CASE eObjectType OF
	E_BACnetObjType.ObjAnalogInput:
		IF ePropID = E_BACnetPropIdentifier.PropPresentValue OR ePropID = E_BACnetPropIdentifier.PropStatusFlags THEN
			F_IsCovProperty:=TRUE;
		END_IF
	E_BACnetObjType.ObjAnalogOutput:
		IF ePropID = E_BACnetPropIdentifier.PropPresentValue OR ePropID = E_BACnetPropIdentifier.PropStatusFlags THEN
			F_IsCovProperty:=TRUE;
		END_IF
	E_BACnetObjType.ObjAnalogValue:
		IF ePropID = E_BACnetPropIdentifier.PropPresentValue OR ePropID = E_BACnetPropIdentifier.PropStatusFlags THEN
			F_IsCovProperty:=TRUE;
		END_IF
	E_BACnetObjType.ObjBinaryInput:
		IF ePropID = E_BACnetPropIdentifier.PropPresentValue OR ePropID = E_BACnetPropIdentifier.PropStatusFlags THEN
			F_IsCovProperty:=TRUE;
		END_IF
	E_BACnetObjType.ObjBinaryOutput:
		IF ePropID = E_BACnetPropIdentifier.PropPresentValue OR ePropID = E_BACnetPropIdentifier.PropStatusFlags THEN
			F_IsCovProperty:=TRUE;
		END_IF
	E_BACnetObjType.ObjBinaryValue:
		IF ePropID = E_BACnetPropIdentifier.PropPresentValue OR ePropID = E_BACnetPropIdentifier.PropStatusFlags THEN
			F_IsCovProperty:=TRUE;
		END_IF
	E_BACnetObjType.ObjMultiStateInput:
		IF ePropID = E_BACnetPropIdentifier.PropPresentValue OR ePropID = E_BACnetPropIdentifier.PropStatusFlags THEN
			F_IsCovProperty:=TRUE;
		END_IF
	E_BACnetObjType.ObjMultiStateOutput:
		IF ePropID = E_BACnetPropIdentifier.PropPresentValue OR ePropID = E_BACnetPropIdentifier.PropStatusFlags THEN
			F_IsCovProperty:=TRUE;
		END_IF
	E_BACnetObjType.ObjMultiStateValue:
		IF ePropID = E_BACnetPropIdentifier.PropPresentValue OR ePropID = E_BACnetPropIdentifier.PropStatusFlags THEN
			F_IsCovProperty:=TRUE;
		END_IF
	E_BACnetObjType.ObjLargeAnalogValue:
		IF ePropID = E_BACnetPropIdentifier.PropPresentValue OR ePropID = E_BACnetPropIdentifier.PropStatusFlags THEN
			F_IsCovProperty:=TRUE;
		END_IF
	E_BACnetObjType.ObjPositiveIntegerValue:
		IF ePropID = E_BACnetPropIdentifier.PropPresentValue OR ePropID = E_BACnetPropIdentifier.PropStatusFlags THEN
			F_IsCovProperty:=TRUE;
		END_IF
	E_BACnetObjType.ObjIntegerValue:
		IF ePropID = E_BACnetPropIdentifier.PropPresentValue OR ePropID = E_BACnetPropIdentifier.PropStatusFlags THEN
			F_IsCovProperty:=TRUE;
		END_IF
	E_BACnetObjType.ObjOctetStringValue:
		IF ePropID = E_BACnetPropIdentifier.PropPresentValue OR ePropID = E_BACnetPropIdentifier.PropStatusFlags THEN
			F_IsCovProperty:=TRUE;
		END_IF
	E_BACnetObjType.ObjCharacterStringValue:
		IF ePropID = E_BACnetPropIdentifier.PropPresentValue OR ePropID = E_BACnetPropIdentifier.PropStatusFlags THEN
			F_IsCovProperty:=TRUE;
		END_IF
	E_BACnetObjType.ObjTimePatternValue:
		IF ePropID = E_BACnetPropIdentifier.PropPresentValue OR ePropID = E_BACnetPropIdentifier.PropStatusFlags THEN
			F_IsCovProperty:=TRUE;
		END_IF
	E_BACnetObjType.ObjTimeValue:
		IF ePropID = E_BACnetPropIdentifier.PropPresentValue OR ePropID = E_BACnetPropIdentifier.PropStatusFlags THEN
			F_IsCovProperty:=TRUE;
		END_IF
	E_BACnetObjType.ObjDatePatternValue:
		IF ePropID = E_BACnetPropIdentifier.PropPresentValue OR ePropID = E_BACnetPropIdentifier.PropStatusFlags THEN
			F_IsCovProperty:=TRUE;
		END_IF
	E_BACnetObjType.ObjDateValue:
		IF ePropID = E_BACnetPropIdentifier.PropPresentValue OR ePropID = E_BACnetPropIdentifier.PropStatusFlags THEN
			F_IsCovProperty:=TRUE;
		END_IF
	E_BACnetObjType.ObjDateTimePatternValue:
		IF ePropID = E_BACnetPropIdentifier.PropPresentValue OR ePropID = E_BACnetPropIdentifier.PropStatusFlags THEN
			F_IsCovProperty:=TRUE;
		END_IF
	E_BACnetObjType.ObjDateTimeValue:
		IF ePropID = E_BACnetPropIdentifier.PropPresentValue OR ePropID = E_BACnetPropIdentifier.PropStatusFlags THEN
			F_IsCovProperty:=TRUE;
		END_IF
	E_BACnetObjType.ObjLoop:
		IF ePropID = E_BACnetPropIdentifier.PropPresentValue OR ePropID = E_BACnetPropIdentifier.PropStatusFlags OR ePropID = E_BACnetPropIdentifier.PropSetpoint OR ePropID = E_BACnetPropIdentifier.PropControlledVariableValue THEN
			F_IsCovProperty:=TRUE;
		END_IF
	E_BACnetObjType.ObjPulseConverter:
			IF ePropID = E_BACnetPropIdentifier.PropPresentValue OR ePropID = E_BACnetPropIdentifier.PropStatusFlags OR ePropID = E_BACnetPropIdentifier.PropUpdateTime THEN
			F_IsCovProperty:=TRUE;
		END_IF
END_CASE

END_FUNCTION

// POUs/Helper/[internal]/Remote/F_IsCovReadMode
{attribute 'hide'}
FUNCTION F_IsCovReadMode : BOOL
VAR_INPUT
	eReadMode : E_BACnet_CommMode;
END_VAR

IF eReadMode = E_BACnet_CommMode.eCov OR eReadMode = E_BACnet_CommMode.eCovC OR eReadMode = E_BACnet_CommMode.eCovU THEN
	F_IsCovReadMode:=TRUE;
END_IF

END_FUNCTION

// POUs/Helper/[internal]/Remote/F_IsCovReqType
{attribute 'hide'}
FUNCTION F_IsCovReqType : BOOL
VAR_INPUT
	iReq : I_BACnetRM_BaseReq;
END_VAR
VAR
	tmpReqType : E_BACnetRM_RequestType;
END_VAR

tmpReqType := iReq.GetRequestType();

IF tmpReqType = E_BACnetRM_RequestType.eCOV OR tmpReqType = E_BACnetRM_RequestType.eCOV_C OR tmpReqType = E_BACnetRM_RequestType.eCOV_U THEN
	F_IsCovReqType:=TRUE;
END_IF

END_FUNCTION

// POUs/Helper/[internal]/Validation-Functions/F_BACnet_IsAbortReasonValid
{attribute 'hide'}
FUNCTION F_BACnet_IsAbortReasonValid : BOOL
VAR_INPUT
	eReason		: E_BACnet_AbortReason;
END_VAR

F_BACnet_IsAbortReasonValid := (E_BACnet_AbortReason.First <= eReason) AND_THEN (eReason <= E_BACnet_AbortReason.Last);

END_FUNCTION

// POUs/Helper/[internal]/Validation-Functions/F_BACnet_IsErrorClassValid
{attribute 'hide'}
FUNCTION F_BACnet_IsErrorClassValid : BOOL
VAR_INPUT
	eClass		: E_BACnet_ErrorClass;
END_VAR

F_BACnet_IsErrorClassValid := (E_BACnet_ErrorClass.First <= eClass) AND_THEN (eClass <= E_BACnet_ErrorClass.Last);

END_FUNCTION

// POUs/Helper/[internal]/Validation-Functions/F_BACnet_IsErrorCodeValid
{attribute 'hide'}
FUNCTION F_BACnet_IsErrorCodeValid : BOOL
VAR_INPUT
	eCode		: E_BACnet_ErrorCode;
END_VAR

F_BACnet_IsErrorCodeValid := (E_BACnet_ErrorCode.First <= eCode) AND_THEN (eCode <= E_BACnet_ErrorCode.Last);

END_FUNCTION

// POUs/Helper/[internal]/Validation-Functions/F_BACnet_IsErrorTypeValid
{attribute 'hide'}
FUNCTION F_BACnet_IsErrorTypeValid : BOOL
VAR_INPUT
	eType		: E_BACnet_ErrorType;
END_VAR

F_BACnet_IsErrorTypeValid := (E_BACnet_ErrorType.First <= eType) AND_THEN (eType <= E_BACnet_ErrorType.Last);

END_FUNCTION

// POUs/Helper/[internal]/Validation-Functions/F_BACnet_IsPropIdentifierValid
{attribute 'hide'}
FUNCTION F_BACnet_IsPropIdentifierValid : BOOL
VAR_INPUT
	eProperty		: E_BACnetPropIdentifier;
END_VAR

F_BACnet_IsPropIdentifierValid := (eProperty <> E_BACnetPropIdentifier.PropInvalid);

END_FUNCTION

// POUs/Helper/[internal]/Validation-Functions/F_BACnet_IsRejectReasonValid
{attribute 'hide'}
FUNCTION F_BACnet_IsRejectReasonValid : BOOL
VAR_INPUT
	eReason		: E_BACnet_RejectReason;
END_VAR

F_BACnet_IsRejectReasonValid := (E_BACnet_RejectReason.First <= eReason) AND_THEN (eReason <= E_BACnet_RejectReason.Last);

END_FUNCTION

// POUs/Helper/[internal]/F_BACnet_AnalogPV
{attribute 'hide'}
FUNCTION F_BACnet_AnalogPV : REAL
VAR_INPUT
	bEnable	: BOOL; (* TRUE = commit to stack, FALSE = do-nothing *)
	bNull	: BOOL; (* TRUE = clear priority, FALSE = write value from input *)
	fValue	: REAL;
END_VAR
VAR
	pres : POINTER TO DWORD;
END_VAR

IF (bEnable) THEN
	IF (bNull) THEN
		pres := ADR(F_BACnet_AnalogPV);
		pres^ := F_BACnet_RealNull(); 
	ELSE
		F_BACnet_AnalogPV := fValue;
	END_IF
ELSE
	F_BACnet_AnalogPV := F_BACnet_NAN();
END_IF

END_FUNCTION

// POUs/Helper/Real/F_BACnet_RealNull
FUNCTION F_BACnet_RealNull : DWORD
(* function that generates <not-a-number> real state *)

F_BACnet_RealNull:=16#7FFF0000;

END_FUNCTION

// POUs/Helper/Real/F_BACnet_NAN
FUNCTION F_BACnet_NAN : REAL
(* function that generates <not-a-number> real state *)
VAR
	res : POINTER TO DWORD;
END_VAR

res:=ADR(F_BACnet_NAN);
res^:=16#7FFFFFFF;

END_FUNCTION

// POUs/Helper/[internal]/F_BACnet_ChangeBitFieldBit
{attribute 'hide'}
FUNCTION F_BACnet_ChangeBitFieldBit : DWORD
VAR_INPUT
	ptrData		: POINTER TO DWORD;
	bitNbr			: INT;
	Value		: BOOL;
END_VAR
VAR
END_VAR

IF (NOT Value) THEN
	ptrData^ := ptrData^ AND NOT (SHR(DWORD#16#00008000,F_BACnet_BitFieldBit(bitNbr)));
ELSE
	ptrData^ := ptrData^ OR (SHR(DWORD#16#00008000,F_BACnet_BitFieldBit(bitNbr)));
END_IF
F_BACnet_ChangeBitFieldBit := ptrData^;

END_FUNCTION

// POUs/Helper/[internal]/F_BACnet_ElemSize
{attribute 'hide'}
FUNCTION F_BACnet_ElemSize : UDINT
VAR_INPUT
	nSize : UDINT;
END_VAR

F_BACnet_ElemSize := (nSize AND 16#7FFFFFFF);

END_FUNCTION

// POUs/Helper/[internal]/F_BACnet_IsBitFieldBitSetPtr
{attribute 'hide'}
FUNCTION F_BACnet_IsBitFieldBitSetPtr : BOOL
VAR_INPUT
	pData	:	POINTER TO WORD;
	bitNbr	:	INT;
END_VAR
VAR
END_VAR

F_BACnet_IsBitFieldBitSetPtr:= ((pData^) AND (SHR(16#8000,F_BACnet_BitFieldBit(bitNbr)))) > 0;

END_FUNCTION

// POUs/Helper/[internal]/F_BACnet_UnSetBitFieldBit
{attribute 'hide'}
FUNCTION F_BACnet_UnSetBitFieldBit : DWORD
VAR_INPUT
	ptrData		:	POINTER TO DWORD;
	bitNbr			:	INT;
END_VAR
VAR
END_VAR

ptrData^ := ptrData^ AND NOT (SHR(DWORD#16#00008000,F_BACnet_BitFieldBit(bitNbr)));
F_BACnet_UnSetBitFieldBit := ptrData^;

END_FUNCTION

// POUs/Helper/Flags/F_BACnet_EventEnable
FUNCTION F_BACnet_EventEnable : UINT
VAR_INPUT
	stEvtEn       : ST_BA_EventTransitions;
END_VAR
VAR
	nEvtEnToFlt     : UINT;
	nEvtEnToNmal    : UINT;
	nEvtEnToOffnmal : UINT;
	nEvtEnNo        : UINT;
END_VAR

(*=============================================*)
(*EventEnable*)
IF	stEvtEn.bToFault
THEN
	nEvtEnToFlt := 16#4000;
ELSE
	nEvtEnToFlt := 16#0;
END_IF

IF	stEvtEn.bToNormal
THEN
	nEvtEnToNmal := 16#2000;
ELSE
	nEvtEnToNmal := 16#0;
END_IF

IF	stEvtEn.bToOffnormal
THEN
	nEvtEnToOffnmal := 16#8000;
ELSE
	nEvtEnToOffnmal := 16#0;
END_IF

nEvtEnNo := 5;

F_BACnet_EventEnable := nEvtEnNo + nEvtEnToFlt + nEvtEnToNmal + nEvtEnToOffnmal;
(*=============================================*)

END_FUNCTION

// POUs/Helper/Flags/F_BACnet_EventTransitionFlags
FUNCTION F_BACnet_EventTransitionFlags : ST_BA_EventTransitions
VAR_INPUT
	data	: WORD;
END_VAR
VAR
END_VAR

F_BACnet_EventTransitionFlags.bToNormal := F_BACnet_IsBitFieldBitSet(data, E_BACnet_EventTransitionBits.eToNormal);
F_BACnet_EventTransitionFlags.bToOffnormal := F_BACnet_IsBitFieldBitSet(data, E_BACnet_EventTransitionBits.eToOffnormal);
F_BACnet_EventTransitionFlags.bToFault := F_BACnet_IsBitFieldBitSet(data, E_BACnet_EventTransitionBits.eToFault);

END_FUNCTION

// POUs/Helper/Flags/F_BACnet_GetEventTransFlagsData
FUNCTION F_BACnet_GetEventTransFlagsData : WORD
VAR_INPUT
	Flags	: ST_BA_EventTransitions;
END_VAR
VAR
END_VAR

F_BACnet_GetEventTransFlagsData := 16#0005;
IF Flags.bToNormal THEN
	F_BACnet_GetEventTransFlagsData := DWORD_TO_WORD(F_BACnet_SetBitFieldBit(ptrData:=ADR(F_BACnet_GetEventTransFlagsData), bitNbr:=E_BACnet_EventTransitionBits.eToNormal));
END_IF
IF Flags.bToOffnormal THEN
	F_BACnet_GetEventTransFlagsData := DWORD_TO_WORD(F_BACnet_SetBitFieldBit(ptrData:=ADR(F_BACnet_GetEventTransFlagsData), bitNbr:=E_BACnet_EventTransitionBits.eToOffnormal));
END_IF
IF Flags.bToFault THEN
	F_BACnet_GetEventTransFlagsData := DWORD_TO_WORD(F_BACnet_SetBitFieldBit(ptrData:=ADR(F_BACnet_GetEventTransFlagsData), bitNbr:=E_BACnet_EventTransitionBits.eToFault));
END_IF

END_FUNCTION

// POUs/Helper/Flags/F_BACnet_GetLimitEnFlagsData
FUNCTION F_BACnet_GetLimitEnFlagsData : WORD
VAR_INPUT
	Flags	: ST_BACnet_LimitEnable;
END_VAR
VAR
END_VAR

F_BACnet_GetLimitEnFlagsData := 16#0006;
IF Flags.highLimitEnable THEN
	F_BACnet_GetLimitEnFlagsData := DWORD_TO_WORD(F_BACnet_SetBitFieldBit(ptrData:=ADR(F_BACnet_GetLimitEnFlagsData), bitNbr:=E_BACnet_LimitEnableBits.eHighLimit));
END_IF
IF Flags.lowLimitEnable THEN
	F_BACnet_GetLimitEnFlagsData := DWORD_TO_WORD(F_BACnet_SetBitFieldBit(ptrData:=ADR(F_BACnet_GetLimitEnFlagsData), bitNbr:=E_BACnet_LimitEnableBits.eLowLimit));
END_IF

END_FUNCTION

// POUs/Helper/Flags/F_BACnet_GetStatusFlagsData
FUNCTION F_BACnet_GetStatusFlagsData : WORD
VAR_INPUT
	Flags : ST_BA_StatusFlags;
END_VAR

(*
F_BACnet_GetStatusFlagsData	:= 16#0004;
IF Flags.bInAlarm THEN
	F_BACnet_GetStatusFlagsData := DWORD_TO_WORD(F_BACnet_SetBitFieldBit(ptrData:=ADR(F_BACnet_GetStatusFlagsData), bitNbr:=E_BACnet_StatusFlags.eInAlarm));
END_IF
IF Flags.bFault THEN
	F_BACnet_GetStatusFlagsData := DWORD_TO_WORD(F_BACnet_SetBitFieldBit(ptrData:=ADR(F_BACnet_GetStatusFlagsData), bitNbr:=E_BACnet_StatusFlags.eFault));
END_IF
IF Flags.bOverridden THEN
	F_BACnet_GetStatusFlagsData := DWORD_TO_WORD(F_BACnet_SetBitFieldBit(ptrData:=ADR(F_BACnet_GetStatusFlagsData), bitNbr:=E_BACnet_StatusFlags.eOverridden));
END_IF
IF Flags.bOutOfService THEN
	F_BACnet_GetStatusFlagsData := DWORD_TO_WORD(F_BACnet_SetBitFieldBit(ptrData:=ADR(F_BACnet_GetStatusFlagsData), bitNbr:=E_BACnet_StatusFlags.eOutOfService));
END_IF
*)

// More performant:
F_BACnet_GetStatusFlagsData		:=	16#0004 +
	TO_WORD(Flags.bInAlarm) 		* 16#8000 +
	TO_WORD(Flags.bFault) 			* 16#4000 +
	TO_WORD(Flags.bOverridden) 		* 16#2000 +
	TO_WORD(Flags.bOutOfService) 	* 16#1000;

END_FUNCTION

// POUs/Helper/Flags/F_BACnet_LimitEnable
FUNCTION F_BACnet_LimitEnable : UINT
VAR_INPUT
	stLimEn         : ST_BACnet_LimitEnable;
END_VAR
VAR
	nHiLimEn     : UINT;
	nLowLimEn    : UINT;
	nLimEnNo     : UINT;
END_VAR

(*=============================================*)
IF	stLimEn.highLimitEnable
THEN
	nHiLimEn := 16#4000;
ELSE
	nHiLimEn := 16#0;
END_IF


IF	stLimEn.lowLimitEnable
THEN
	nLowLimEn := 16#8000;
ELSE
	nLowLimEn := 16#0;
END_IF

nLimEnNo := 16#6;

F_BACnet_LimitEnable := nLimEnNo + nHiLimEn + nLowLimEn;
(*=============================================*)

END_FUNCTION

// POUs/Helper/Flags/F_BACnet_LimitEnableFlags
FUNCTION F_BACnet_LimitEnableFlags : ST_BACnet_LimitEnable
VAR_INPUT
	data	: WORD;
END_VAR
VAR
END_VAR

F_BACnet_LimitEnableFlags.highLimitEnable := F_BACnet_IsBitFieldBitSet( data:=data, bitNbr:=E_BACnet_LimitEnableBits.eHighLimit);
F_BACnet_LimitEnableFlags.lowLimitEnable := F_BACnet_IsBitFieldBitSet( data:=data, bitNbr:=E_BACnet_LimitEnableBits.eLowLimit);

END_FUNCTION

// POUs/Helper/Flags/F_BACnet_StatusFlags
FUNCTION F_BACnet_StatusFlags : ST_BA_StatusFlags
VAR_INPUT
	data	: WORD;
END_VAR
VAR
END_VAR

F_BACnet_StatusFlags.bInAlarm:= F_BACnet_IsBitFieldBitSet( data:=data, bitNbr:=E_BACnet_StatusFlags.eInAlarm);
F_BACnet_StatusFlags.bFault:= F_BACnet_IsBitFieldBitSet( data:=data, bitNbr:=E_BACnet_StatusFlags.eFault);
F_BACnet_StatusFlags.bOverridden:= F_BACnet_IsBitFieldBitSet( data:=data, bitNbr:=E_BACnet_StatusFlags.eOverridden);
F_BACnet_StatusFlags.bOutOfService:= F_BACnet_IsBitFieldBitSet( data:=data, bitNbr:=E_BACnet_StatusFlags.eOutOfService);

END_FUNCTION

// POUs/Helper/MultiState/F_BACnet_EnMultiStatePV
FUNCTION F_BACnet_EnMultiStatePV : UDINT
VAR_INPUT
	bEnable			: BOOL;
	nValue			: UDINT;
END_VAR

IF (bEnable) THEN
	F_BACnet_EnMultiStatePV := MAX(nValue, E_BACnet_MultistateVal.eMin);
ELSE
	F_BACnet_EnMultiStatePV := E_BACnet_MultistateVal.eNull;
END_IF

END_FUNCTION

// POUs/Helper/MultiState/F_BACnet_MultiStatePV
FUNCTION F_BACnet_MultiStatePV : UDINT
VAR_INPUT
	bEnable						: BOOL; (* TRUE = commit to stack, FALSE = do-nothing *)
	bNull						: BOOL; (* TRUE = clear priority, FALSE = write number from state input *)
	nState						: UDINT; (* multi-state [1..max-number-of-states] *)
END_VAR

IF (bEnable) THEN
	IF (bNull) THEN
		F_BACnet_MultiStatePV := E_BACnet_MultistateVal.eNull;
	ELSE
		F_BACnet_MultiStatePV := MAX(nState, E_BACnet_MultistateVal.eMin);
	END_IF
ELSE
	F_BACnet_MultiStatePV := E_BACnet_MultistateVal.eNothing;
END_IF

END_FUNCTION

// POUs/Helper/NC/F_BACnet_DeviceRecipient
// Returns an initialized recipient structure.
FUNCTION F_BACnet_DeviceRecipient : ST_BACnet_Recipient
VAR_INPUT
	nDeviceInstance		: UDINT			:= BACnet_Globals.nBACnetInstId_Auto;
END_VAR

F_BACnet_DeviceRecipient.eRecipientChoice := E_BACnet_RecipientChoice.eDevice;
F_BACnet_DeviceRecipient.stEntry.nDeviceInstance := F_BACnet_GetObjId(E_BACnetObjType.ObjDevice,nDeviceInstance);

END_FUNCTION

// POUs/Helper/NC/F_BACnet_EthernetRecipient
// Returns an initialized recipient structure.
FUNCTION F_BACnet_EthernetRecipient : ST_BACnet_Recipient
VAR_INPUT
	nIPAddress1		: BYTE;
	nIPAddress2		: BYTE;
	nIPAddress3		: BYTE;
	nIPAddress4		: BYTE;
	nPort			: UINT;
	nNetworkNr		: UINT;
END_VAR
VAR
	_nPort			: POINTER TO ARRAY[0 .. 1] OF BYTE := ADR(nPort);
END_VAR

F_BACnet_EthernetRecipient.eRecipientChoice := E_BACnet_RecipientChoice.eAddress;
F_BACnet_EthernetRecipient.stEntry.stNetAddr.eChoice := E_BACnet_AddressChoice.eEthernet;
F_BACnet_EthernetRecipient.stEntry.stNetAddr.nNetworkNr := nNetworkNr;
F_BACnet_EthernetRecipient.stEntry.stNetAddr.aAddress[0] := nIPAddress1;
F_BACnet_EthernetRecipient.stEntry.stNetAddr.aAddress[1] := nIPAddress2;
F_BACnet_EthernetRecipient.stEntry.stNetAddr.aAddress[2] := nIPAddress3;
F_BACnet_EthernetRecipient.stEntry.stNetAddr.aAddress[3] := nIPAddress4;

// Swap Port-Bytes:
F_BACnet_EthernetRecipient.stEntry.stNetAddr.aAddress[4] := _nPort^[1];
F_BACnet_EthernetRecipient.stEntry.stNetAddr.aAddress[5] := _nPort^[0];

END_FUNCTION

// POUs/Helper/NC/F_BACnet_EthernetRecipientEx
// Returns an initialized recipient structure.
FUNCTION F_BACnet_EthernetRecipientEx : ST_BACnet_Recipient
VAR_INPUT
	tIPAddress		: T_IPv4AddrArr;
	nPort			: UINT;
	nNetworkNr		: UINT;
END_VAR

F_BACnet_EthernetRecipientEx := F_BACnet_EthernetRecipient(tIPAddress[0], tIPAddress[1], tIPAddress[2], tIPAddress[3], nPort, nNetworkNr);

END_FUNCTION

// POUs/Helper/Real/F_BACnet_EnRealPV
FUNCTION F_BACnet_EnRealPV : DWORD
VAR_INPUT
	bEnable	: BOOL;
	fValue	: REAL;
END_VAR
VAR
	pDword : POINTER TO DWORD;
END_VAR

IF (bEnable) THEN
	pDword := ADR(fValue);
	F_BACnet_EnRealPV := pDword^;
ELSE
	F_BACnet_EnRealPV := F_BACnet_RealNull();
END_IF

END_FUNCTION

// POUs/Helper/Real/F_BACnet_IsFinite
FUNCTION F_BACnet_IsFinite : BOOL
VAR_INPUT
	fValue		: REAL;
END_VAR
VAR
	fArg		: T_Arg;
END_VAR

fArg.cbLen := SIZEOF(fValue);
fArg.eType := ARGTYPE_REAL;
fArg.pData := ADR(fValue);
F_BACnet_IsFinite := IsFinite(fArg);

END_FUNCTION

// POUs/Helper/Real/F_BACnet_RealEQ
FUNCTION F_BACnet_RealEQ : BOOL
VAR_INPUT
	fIn1	: REAL;
	fIn2	: REAL;
END_VAR
VAR
END_VAR

IF (F_BACnet_IsFinite(fIn1) <> F_BACnet_IsFinite(fIn2)) THEN
	F_BACnet_RealEQ := FALSE;
	RETURN;
END_IF
IF F_BACnet_IsFinite(fIn1) THEN
	IF (fIn1 <> fIn2) THEN
		F_BACnet_RealEQ := FALSE;
		RETURN;
	END_IF
END_IF
F_BACnet_RealEQ := TRUE;

END_FUNCTION

// POUs/Helper/Real/F_BACnet_RealGE
FUNCTION F_BACnet_RealGE : BOOL
VAR_INPUT
	fIn1	: REAL;
	fIn2	: REAL;
END_VAR
VAR
END_VAR

IF NOT (F_BACnet_IsFinite(fIn1) OR F_BACnet_IsFinite(fIn2)) THEN
	F_BACnet_RealGE := FALSE;
	RETURN;
END_IF
F_BACnet_RealGE := (fIn1 >= fIn2);

END_FUNCTION

// POUs/Helper/Real/F_BACnet_RealGT
FUNCTION F_BACnet_RealGT : BOOL
VAR_INPUT
	fIn1	: REAL;
	fIn2	: REAL;
END_VAR
VAR
END_VAR

IF NOT (F_BACnet_IsFinite(fIn1) OR F_BACnet_IsFinite(fIn2)) THEN
	F_BACnet_RealGT := FALSE;
	RETURN;
END_IF
F_BACnet_RealGT := (fIn1 > fIn2);

END_FUNCTION

// POUs/Helper/Real/F_BACnet_RealLE
FUNCTION F_BACnet_RealLE : BOOL
VAR_INPUT
	fIn1	: REAL;
	fIn2	: REAL;
END_VAR
VAR
END_VAR

IF NOT (F_BACnet_IsFinite(fIn1) OR F_BACnet_IsFinite(fIn2)) THEN
	F_BACnet_RealLE := FALSE;
	RETURN;
END_IF
F_BACnet_RealLE := (fIn1 <= fIn2);

END_FUNCTION

// POUs/Helper/Real/F_BACnet_RealLT
FUNCTION F_BACnet_RealLT : BOOL
VAR_INPUT
	fIn1	: REAL;
	fIn2	: REAL;
END_VAR
VAR
END_VAR

IF NOT (F_BACnet_IsFinite(fIn1) OR F_BACnet_IsFinite(fIn2)) THEN
	F_BACnet_RealLT := FALSE;
	RETURN;
END_IF
F_BACnet_RealLT := (fIn1 < fIn2);

END_FUNCTION

// POUs/Helper/Real/F_BACnet_RealNothing
FUNCTION F_BACnet_RealNothing : DWORD

F_BACnet_RealNothing:=16#7FFFFFFF;

END_FUNCTION

// POUs/Helper/Real/F_BACnet_RealPV
FUNCTION F_BACnet_RealPV : DWORD
VAR_INPUT
	bEnable	: BOOL; (* TRUE = commit to stack, FALSE = do-nothing *)
	bNull	: BOOL; (* TRUE = clear priority, FALSE = write value from input *)
	fValue	: REAL;
END_VAR
VAR
	pDword : POINTER TO DWORD;
END_VAR

IF (bEnable) THEN
	IF (bNull) THEN
		F_BACnet_RealPV := F_BACnet_RealNull();
	ELSE
		pDword := ADR(fValue);
		F_BACnet_RealPV := pDword^;
	END_IF
ELSE
	F_BACnet_RealPV := F_BACnet_RealNothing();
END_IF

END_FUNCTION

// POUs/Helper/Real/F_BACnet_RealToStr
FUNCTION F_BACnet_RealToStr : STRING
VAR_INPUT
	pValue	: POINTER TO REAL;
END_VAR
VAR
	fArg	: T_Arg;
	pDWORD	: POINTER TO DWORD;
END_VAR

IF (pValue <> 0) THEN
	fArg.cbLen := 4;
	fArg.eType := ARGTYPE_REAL;
	fArg.pData := pValue;
	pDWORD := pValue;
	IF IsFinite(fArg) THEN
		F_BACnet_RealToStr := REAL_TO_STRING(pValue^);
	ELSE
		IF (pDWORD^ = 16#7FFF0000) THEN
			F_BACnet_RealToStr := '#NULL';
		ELSIF (pDWORD^ AND 16#80000000) = 16#80000000 THEN
			F_BACnet_RealToStr := '-#QNAN';
		ELSE
			F_BACnet_RealToStr := '#QNAN';
		END_IF
	END_IF
END_IF

END_FUNCTION

// POUs/Helper/References/F_BACnet_Reference
FUNCTION F_BACnet_Reference : ST_BACnet_ObjectPropertyReference
VAR_INPUT
	iObject				: I_BACnet_Object;
	ePropertyId			: E_BACnetPropIdentifier		:= E_BACnetPropIdentifier.PropPresentValue;
END_VAR

F_BACnet_Reference.iObject := iObject;
F_BACnet_Reference.tObjectID := BACnet_Globals.nBACnetObjId_None;
F_BACnet_Reference.ePropertyId := ePropertyId;

END_FUNCTION

// POUs/Helper/References/F_BACnet_ReferenceByID
FUNCTION F_BACnet_ReferenceByID : ST_BACnet_ObjectPropertyReference
VAR_INPUT
	tObjectID			: T_BACnet_ObjectIdentifier;
	ePropertyId			: E_BACnetPropIdentifier		:= E_BACnetPropIdentifier.PropPresentValue;
END_VAR

F_BACnet_ReferenceByID.iObject := 0;
F_BACnet_ReferenceByID.tObjectID := tObjectID;
F_BACnet_ReferenceByID.ePropertyId := ePropertyId;

END_FUNCTION

// POUs/Helper/Schedule/Calendar/F_BACnet_SchedCalendar
// Returns an initialized analog weekly scheduler.
FUNCTION F_BACnet_SchedCalendar : T_BACnet_SchedCalendar
VAR_INPUT
	iRefCalendar1	: I_BACnet_Cal	:= 0;
	iRefCalendar2	: I_BACnet_Cal	:= 0;
	iRefCalendar3	: I_BACnet_Cal	:= 0;
END_VAR
VAR
	nIndex			: INT;
END_VAR

F_BACnet_SchedCalendar[1].iRefCalendar := iRefCalendar1;

nIndex := 2;
IF (BACnet_Param.nSched_CalendarCount >= nIndex) THEN
	F_BACnet_SchedCalendar[nIndex].iRefCalendar := iRefCalendar2;
END_IF

nIndex := 3;
IF (BACnet_Param.nSched_CalendarCount >= nIndex) THEN
	F_BACnet_SchedCalendar[nIndex].iRefCalendar := iRefCalendar3;
END_IF

END_FUNCTION

// POUs/Helper/Schedule/Exception/F_BACnet_SchedEntry1xA
// Returns an initialized analog weekly scheduler.
FUNCTION F_BACnet_SchedEntry1xA : T_BACnet_SchedExceptionEntryList
VAR_INPUT
	tTime1		: TIME;
	fValue1		: REAL;
END_VAR

F_BA_SetSchedulerEntry(F_BACnet_SchedEntry1xA[1], tTime1, F_BA_RVal(fValue1));

END_FUNCTION

// POUs/Helper/Schedule/Exception/F_BACnet_SchedEntry1xB
// Returns an initialized binary weekly scheduler.
FUNCTION F_BACnet_SchedEntry1xB : T_BACnet_SchedExceptionEntryList
VAR_INPUT
	tTime1		: TIME;
	bValue1		: BOOL;
END_VAR

F_BA_SetSchedulerEntry(F_BACnet_SchedEntry1xB[1], tTime1, F_BA_BVal(bValue1));

END_FUNCTION

// POUs/Helper/Schedule/Exception/F_BACnet_SchedEntry1xM
// Returns an initialized multistate weekly scheduler.
FUNCTION F_BACnet_SchedEntry1xM : T_BACnet_SchedExceptionEntryList
VAR_INPUT
	tTime1		: TIME;
	nValue1		: UDINT;
END_VAR

F_BA_SetSchedulerEntry(F_BACnet_SchedEntry1xM[1], tTime1, F_BA_UDIVal(nValue1));

END_FUNCTION

// POUs/Helper/Schedule/Exception/F_BACnet_SchedEntry3xA
// Returns an initialized analog weekly scheduler.
FUNCTION F_BACnet_SchedEntry3xA : T_BACnet_SchedExceptionEntryList
VAR_INPUT
	tTime1		: TIME;
	fValue1		: REAL;
	tTime2		: TIME;
	fValue2		: REAL;
	tTime3		: TIME;
	fValue3		: REAL;
END_VAR

F_BA_SetSchedulerEntry(F_BACnet_SchedEntry3xA[1], tTime1, F_BA_RVal(fValue1));
F_BA_SetSchedulerEntry(F_BACnet_SchedEntry3xA[2], tTime2, F_BA_RVal(fValue2));
F_BA_SetSchedulerEntry(F_BACnet_SchedEntry3xA[3], tTime3, F_BA_RVal(fValue3));

END_FUNCTION

// POUs/Helper/Schedule/Exception/F_BACnet_SchedEntry3xB
// Returns an initialized binary weekly scheduler.
FUNCTION F_BACnet_SchedEntry3xB : T_BACnet_SchedExceptionEntryList
VAR_INPUT
	tTime1		: TIME;
	bValue1		: BOOL;
	tTime2		: TIME;
	bValue2		: BOOL;
	tTime3		: TIME;
	bValue3		: BOOL;
END_VAR

F_BA_SetSchedulerEntry(F_BACnet_SchedEntry3xB[1], tTime1, F_BA_BVal(bValue1));
F_BA_SetSchedulerEntry(F_BACnet_SchedEntry3xB[2], tTime2, F_BA_BVal(bValue2));
F_BA_SetSchedulerEntry(F_BACnet_SchedEntry3xB[3], tTime3, F_BA_BVal(bValue3));

END_FUNCTION

// POUs/Helper/Schedule/Exception/F_BACnet_SchedEntry3xM
// Returns an initialized multistate weekly scheduler.
FUNCTION F_BACnet_SchedEntry3xM : T_BACnet_SchedExceptionEntryList
VAR_INPUT
	tTime1		: TIME;
	nValue1		: UDINT;
	tTime2		: TIME;
	nValue2		: UDINT;
	tTime3		: TIME;
	nValue3		: UDINT;
END_VAR

F_BA_SetSchedulerEntry(F_BACnet_SchedEntry3xM[1], tTime1, F_BA_UDIVal(nValue1));
F_BA_SetSchedulerEntry(F_BACnet_SchedEntry3xM[2], tTime2, F_BA_UDIVal(nValue2));
F_BA_SetSchedulerEntry(F_BACnet_SchedEntry3xM[3], tTime3, F_BA_UDIVal(nValue3));

END_FUNCTION

// POUs/Helper/Schedule/Exception/F_BACnet_SchedEntry5xA
// Returns an initialized analog weekly scheduler.
FUNCTION F_BACnet_SchedEntry5xA : T_BACnet_SchedExceptionEntryList
VAR_INPUT
	tTime1		: TIME;
	fValue1		: REAL;
	tTime2		: TIME;
	fValue2		: REAL;
	tTime3		: TIME;
	fValue3		: REAL;
	tTime4		: TIME;
	fValue4		: REAL;
	tTime5		: TIME;
	fValue5		: REAL;
END_VAR

F_BA_SetSchedulerEntry(F_BACnet_SchedEntry5xA[1], tTime1, F_BA_RVal(fValue1));
F_BA_SetSchedulerEntry(F_BACnet_SchedEntry5xA[2], tTime2, F_BA_RVal(fValue2));
F_BA_SetSchedulerEntry(F_BACnet_SchedEntry5xA[3], tTime3, F_BA_RVal(fValue3));
F_BA_SetSchedulerEntry(F_BACnet_SchedEntry5xA[4], tTime4, F_BA_RVal(fValue4));
F_BA_SetSchedulerEntry(F_BACnet_SchedEntry5xA[5], tTime5, F_BA_RVal(fValue5));

END_FUNCTION

// POUs/Helper/Schedule/Exception/F_BACnet_SchedEntry5xB
// Returns an initialized binary weekly scheduler.
FUNCTION F_BACnet_SchedEntry5xB : T_BACnet_SchedExceptionEntryList
VAR_INPUT
	tTime1		: TIME;
	bValue1		: BOOL;
	tTime2		: TIME;
	bValue2		: BOOL;
	tTime3		: TIME;
	bValue3		: BOOL;
	tTime4		: TIME;
	bValue4		: BOOL;
	tTime5		: TIME;
	bValue5		: BOOL;
END_VAR

F_BA_SetSchedulerEntry(F_BACnet_SchedEntry5xB[1], tTime1, F_BA_BVal(bValue1));
F_BA_SetSchedulerEntry(F_BACnet_SchedEntry5xB[2], tTime2, F_BA_BVal(bValue2));
F_BA_SetSchedulerEntry(F_BACnet_SchedEntry5xB[3], tTime3, F_BA_BVal(bValue3));
F_BA_SetSchedulerEntry(F_BACnet_SchedEntry5xB[4], tTime4, F_BA_BVal(bValue4));
F_BA_SetSchedulerEntry(F_BACnet_SchedEntry5xB[5], tTime5, F_BA_BVal(bValue5));

END_FUNCTION

// POUs/Helper/Schedule/Exception/F_BACnet_SchedEntry5xM
// Returns an initialized multistate weekly scheduler.
FUNCTION F_BACnet_SchedEntry5xM : T_BACnet_SchedExceptionEntryList
VAR_INPUT
	tTime1		: TIME;
	nValue1		: UDINT;
	tTime2		: TIME;
	nValue2		: UDINT;
	tTime3		: TIME;
	nValue3		: UDINT;
	tTime4		: TIME;
	nValue4		: UDINT;
	tTime5		: TIME;
	nValue5		: UDINT;
END_VAR

F_BA_SetSchedulerEntry(F_BACnet_SchedEntry5xM[1], tTime1, F_BA_UDIVal(nValue1));
F_BA_SetSchedulerEntry(F_BACnet_SchedEntry5xM[2], tTime2, F_BA_UDIVal(nValue2));
F_BA_SetSchedulerEntry(F_BACnet_SchedEntry5xM[3], tTime3, F_BA_UDIVal(nValue3));
F_BA_SetSchedulerEntry(F_BACnet_SchedEntry5xM[4], tTime4, F_BA_UDIVal(nValue4));
F_BA_SetSchedulerEntry(F_BACnet_SchedEntry5xM[5], tTime5, F_BA_UDIVal(nValue5));

END_FUNCTION

// POUs/Helper/Schedule/Weekly/F_BACnet_SchedWeekly3xA
// Returns an initialized analog weekly scheduler.
FUNCTION F_BACnet_SchedWeekly3xA : T_BACnet_SchedWeek
VAR_INPUT
	eDayFrom	: E_BA_Weekday		:= E_BA_Weekday.eMonday;
	eDayTo		: E_BA_Weekday		:= E_BA_Weekday.eSunday;
	
	tTime1		: TIME;
	fValue1		: REAL;
	tTime2		: TIME;
	fValue2		: REAL;
	tTime3		: TIME;
	fValue3		: REAL;
END_VAR

F_BA_SetWeekdays(F_BACnet_SchedWeekly3xA, eDayFrom, eDayTo, 1, tTime1, F_BA_RVal(fValue1));
F_BA_SetWeekdays(F_BACnet_SchedWeekly3xA, eDayFrom, eDayTo, 2, tTime2, F_BA_RVal(fValue2));
F_BA_SetWeekdays(F_BACnet_SchedWeekly3xA, eDayFrom, eDayTo, 3, tTime3, F_BA_RVal(fValue3));

END_FUNCTION

// POUs/Helper/Schedule/Weekly/F_BACnet_SchedWeekly3xB
// Returns an initialized binary weekly scheduler.
FUNCTION F_BACnet_SchedWeekly3xB : T_BACnet_SchedWeek
VAR_INPUT
	eDayFrom	: E_BA_Weekday		:= E_BA_Weekday.eMonday;
	eDayTo		: E_BA_Weekday		:= E_BA_Weekday.eSunday;
	
	tTime1		: TIME;
	bValue1		: BOOL;
	tTime2		: TIME;
	bValue2		: BOOL;
	tTime3		: TIME;
	bValue3		: BOOL;
END_VAR

F_BA_SetWeekdays(F_BACnet_SchedWeekly3xB, eDayFrom, eDayTo, 1, tTime1, F_BA_BVal(bValue1));
F_BA_SetWeekdays(F_BACnet_SchedWeekly3xB, eDayFrom, eDayTo, 2, tTime2, F_BA_BVal(bValue2));
F_BA_SetWeekdays(F_BACnet_SchedWeekly3xB, eDayFrom, eDayTo, 3, tTime3, F_BA_BVal(bValue3));

END_FUNCTION

// POUs/Helper/Schedule/Weekly/F_BACnet_SchedWeekly3xM
// Returns an initialized multistate weekly scheduler.
FUNCTION F_BACnet_SchedWeekly3xM : T_BACnet_SchedWeek
VAR_INPUT
	eDayFrom	: E_BA_Weekday		:= E_BA_Weekday.eMonday;
	eDayTo		: E_BA_Weekday		:= E_BA_Weekday.eSunday;
	
	tTime1		: TIME;
	nValue1		: UDINT;
	tTime2		: TIME;
	nValue2		: UDINT;
	tTime3		: TIME;
	nValue3		: UDINT;
END_VAR

F_BA_SetWeekdays(F_BACnet_SchedWeekly3xM, eDayFrom, eDayTo, 1, tTime1, F_BA_UDIVal(nValue1));
F_BA_SetWeekdays(F_BACnet_SchedWeekly3xM, eDayFrom, eDayTo, 2, tTime2, F_BA_UDIVal(nValue2));
F_BA_SetWeekdays(F_BACnet_SchedWeekly3xM, eDayFrom, eDayTo, 3, tTime3, F_BA_UDIVal(nValue3));

END_FUNCTION

// POUs/Helper/Schedule/Weekly/F_BACnet_SchedWeekly5xA
// Returns an initialized analog weekly scheduler.
FUNCTION F_BACnet_SchedWeekly5xA : T_BACnet_SchedWeek
VAR_INPUT
	eDayFrom	: E_BA_Weekday		:= E_BA_Weekday.eMonday;
	eDayTo		: E_BA_Weekday		:= E_BA_Weekday.eSunday;
	
	tTime1		: TIME;
	fValue1		: REAL;
	tTime2		: TIME;
	fValue2		: REAL;
	tTime3		: TIME;
	fValue3		: REAL;
	tTime4		: TIME;
	fValue4		: REAL;
	tTime5		: TIME;
	fValue5		: REAL;
END_VAR

F_BA_SetWeekdays(F_BACnet_SchedWeekly5xA, eDayFrom, eDayTo, 1, tTime1, F_BA_RVal(fValue1));
F_BA_SetWeekdays(F_BACnet_SchedWeekly5xA, eDayFrom, eDayTo, 2, tTime2, F_BA_RVal(fValue2));
F_BA_SetWeekdays(F_BACnet_SchedWeekly5xA, eDayFrom, eDayTo, 3, tTime3, F_BA_RVal(fValue3));
F_BA_SetWeekdays(F_BACnet_SchedWeekly5xA, eDayFrom, eDayTo, 4, tTime4, F_BA_RVal(fValue4));
F_BA_SetWeekdays(F_BACnet_SchedWeekly5xA, eDayFrom, eDayTo, 5, tTime5, F_BA_RVal(fValue5));

END_FUNCTION

// POUs/Helper/Schedule/Weekly/F_BACnet_SchedWeekly5xB
// Returns an initialized binary weekly scheduler.
FUNCTION F_BACnet_SchedWeekly5xB : T_BACnet_SchedWeek
VAR_INPUT
	eDayFrom	: E_BA_Weekday		:= E_BA_Weekday.eMonday;
	eDayTo		: E_BA_Weekday		:= E_BA_Weekday.eSunday;
	
	tTime1		: TIME;
	bValue1		: BOOL;
	tTime2		: TIME;
	bValue2		: BOOL;
	tTime3		: TIME;
	bValue3		: BOOL;
	tTime4		: TIME;
	bValue4		: BOOL;
	tTime5		: TIME;
	bValue5		: BOOL;
END_VAR

F_BA_SetWeekdays(F_BACnet_SchedWeekly5xB, eDayFrom, eDayTo, 1, tTime1, F_BA_BVal(bValue1));
F_BA_SetWeekdays(F_BACnet_SchedWeekly5xB, eDayFrom, eDayTo, 2, tTime2, F_BA_BVal(bValue2));
F_BA_SetWeekdays(F_BACnet_SchedWeekly5xB, eDayFrom, eDayTo, 3, tTime3, F_BA_BVal(bValue3));
F_BA_SetWeekdays(F_BACnet_SchedWeekly5xB, eDayFrom, eDayTo, 4, tTime4, F_BA_BVal(bValue4));
F_BA_SetWeekdays(F_BACnet_SchedWeekly5xB, eDayFrom, eDayTo, 5, tTime5, F_BA_BVal(bValue5));

END_FUNCTION

// POUs/Helper/Schedule/Weekly/F_BACnet_SchedWeekly5xM
// Returns an initialized multistate weekly scheduler.
FUNCTION F_BACnet_SchedWeekly5xM : T_BACnet_SchedWeek
VAR_INPUT
	eDayFrom	: E_BA_Weekday		:= E_BA_Weekday.eMonday;
	eDayTo		: E_BA_Weekday		:= E_BA_Weekday.eSunday;
	
	tTime1		: TIME;
	nValue1		: UDINT;
	tTime2		: TIME;
	nValue2		: UDINT;
	tTime3		: TIME;
	nValue3		: UDINT;
	tTime4		: TIME;
	nValue4		: UDINT;
	tTime5		: TIME;
	nValue5		: UDINT;
END_VAR

F_BA_SetWeekdays(F_BACnet_SchedWeekly5xM, eDayFrom, eDayTo, 1, tTime1, F_BA_UDIVal(nValue1));
F_BA_SetWeekdays(F_BACnet_SchedWeekly5xM, eDayFrom, eDayTo, 2, tTime2, F_BA_UDIVal(nValue2));
F_BA_SetWeekdays(F_BACnet_SchedWeekly5xM, eDayFrom, eDayTo, 3, tTime3, F_BA_UDIVal(nValue3));
F_BA_SetWeekdays(F_BACnet_SchedWeekly5xM, eDayFrom, eDayTo, 4, tTime4, F_BA_UDIVal(nValue4));
F_BA_SetWeekdays(F_BACnet_SchedWeekly5xM, eDayFrom, eDayTo, 5, tTime5, F_BA_UDIVal(nValue5));

END_FUNCTION

// POUs/Helper/String/F_BACnet_GetObjectIdString
FUNCTION F_BACnet_GetObjectIdString : STRING
VAR_INPUT
	tObjectID : T_BACnet_ObjectIdentifier := 16#FFFFFFFF;
END_VAR
VAR
	nObjType	: DINT;
	nObjInstance: UDINT;
END_VAR

nObjType	:= F_BACnet_GetObjType(tObjectID);
nObjInstance:= F_BACnet_GetObjInstance(tObjectID);
IF (BACnet_Globals.nRange_ObjectTypeFirst <= nObjType) AND (nObjType <= BACnet_Globals.nRange_ObjectTypeLast) THEN
	F_BACnet_GetObjectIdString := CONCAT(CONCAT(BACnet_Globals.aSpec_ObjectTypeShortcut[nObjType], ':'), UDINT_TO_STRING(nObjInstance));
ELSE
	F_BACnet_GetObjectIdString := CONCAT('???:', UDINT_TO_STRING(nObjInstance));
END_IF

END_FUNCTION

// POUs/Helper/String/FB_BACnet_StringExtEncode
FUNCTION_BLOCK FB_BACnet_StringExtEncode (* convert Windows-1252 to ANSI/UTF-8 BACnet Character String *)
VAR_INPUT
	pString			: POINTER TO T_MaxString; (* pointer to Windows-1252 encoded PLC text *)
	nSize			: INT; (* string length or data size of pText field *)
	pResultExtStr	: POINTER TO ST_BACnet_CharacterStringExt;
	nResult		: UDINT; (* byte size of result data field *)
END_VAR
VAR_OUTPUT
	bValid			: BOOL;
	bOverflow		: BOOL; (* String length overflow (source string too long) *)
	nLength			: UDINT; (* out string data length in byte *)
END_VAR

(* preset valid to FALSE *)
bOverflow := FALSE;
bValid := TRUE;
(* check pointer *)
IF (pString = 0) OR (pResultExtStr = 0) THEN
	nLength := 0;
	bValid := FALSE;
	RETURN;
END_IF

(* clear string *)
MEMSET(destAddr:=pResultExtStr, fillByte:=0, n:=nResult);
(* check input size *)
IF (nSize <= 0) THEN
	nLength := 0;

(* convert *)
ELSE
	IF (F_BACnet_EncodeUTF8(
		pString		:= pString,
		nString	:= TO_UDINT(nSize),
		pResult		:= pResultExtStr,
		nResult	:= nResult,
		nResultLen	:= nLength) > nResult)
	THEN
		bOverflow	:= TRUE;
		bValid		:= FALSE;
	END_IF
END_IF

END_FUNCTION_BLOCK

// POUs/Helper/F_BACnet_GetObjectListIndex
FUNCTION F_BACnet_GetObjectListIndex : DINT
VAR_INPUT
	tObjectId	: T_BACnet_ObjectIdentifier := 16#FFFFFFFF;
END_VAR

VAR
	nMax : DINT;
	i : DINT;
END_VAR
(*All VAR_IN_OUT variables have been moved to the end of the declaration due to compatibility reasons*)
VAR_IN_OUT
	stObjIDList	: ST_BACnet_ObjectIdentifierList;
END_VAR

nMax := UDINT_TO_DINT(stObjIDList.nEntries)-1;
F_BACnet_GetObjectListIndex := -1; (* preset: no match *)
FOR i := 0 TO nMax DO
	IF stObjIDList.aObjList[i] = tObjectId THEN
		F_BACnet_GetObjectListIndex := i; (* match *)
		RETURN;
	END_IF
END_FOR

END_FUNCTION

// POUs/Helper/FB_BACnet_AvgValue
FUNCTION_BLOCK FB_BACnet_AvgValue
VAR_INPUT
	X	: REAL; (* input value to average *)
	n	: UINT; (* number of averages (0 = no average --> Y = X) *)
END_VAR
VAR_OUTPUT
	Y	: REAL; (* average result *)
END_VAR
VAR
	_n	: UINT := 0;
	_Xn : LREAL;
END_VAR

IF (_n > n) THEN
	_n := n;
END_IF
IF (_n = 0) OR (n = 0) THEN
	_Xn := REAL_TO_LREAL(X);
ELSE
	_Xn := ((_Xn * _n) + REAL_TO_LREAL(X)) / UINT_TO_LREAL(_n + 1);
END_IF
_n := _n + 1;
Y := LREAL_TO_REAL(_Xn);

END_FUNCTION_BLOCK

// POUs/Helper/FB_BACnet_PidControl
FUNCTION_BLOCK FB_BACnet_PidControl
VAR_INPUT
	(* controller input  *)
	fSetpoint				: REAL;	(* setpoint value *)
	fPresentValue			: REAL;	(* actual value *)
	(* reset flag *)
	bReset					: BOOL;
	(* controller values *)
	fCtrlCycleTime			: REAL; (* controller cycle time in seconds [s] *)

	fBias					: REAL; (* bias also active when reset is set to 1 *)
	fKp						: REAL;	(* proportional gain Kp	(P) *)
	fKi						: REAL; (* integral gain Ki (I) *)
	fKd						: REAL;	(* derivative gain Kd (D) *)
	fTp						: REAL := -1.0;	(* damping time Tp (PT1) [s] (fTp < 0 --> Tp = Kd / 10) *)

	(* maximum ratings *)
	fMaxOutput				: REAL;
	fMinOutput				: REAL;
END_VAR
VAR_OUTPUT
	fY						: REAL; (* controller output command *)
	eErrorStatus			: E_BACnet_Error;
END_VAR
VAR
	(* Internal Variable *)
	_fE		: REAL;
	_fEOld	: REAL;
	_fYp	: REAL;
	_fYi	: REAL;
	_fYd	: REAL;
	_fbYd	: FB_BACnet_PT1;
END_VAR

(* preset error number *)
eErrorStatus	:= E_BACnet_Error.eNoError;

(* check cycle time parameter: (CycleTime > 0) *)
IF (fCtrlCycleTime <= 0.0) THEN
	eErrorStatus := E_BACnet_Error.eInvalidCycleTime;
	bReset := TRUE;
END_IF;

(* check controller parameters: (Kp, Ki, Kd >= 0) *)
IF ((fKp < 0.0) OR (fKi < 0.0) OR (fKd < 0.0)) THEN
	eErrorStatus := E_BACnet_Error.eInvalidParameter;
	bReset := TRUE;
END_IF;

(* controller reset *)
IF bReset THEN
	(* reset internal and external variables *)
	_fEOld	:= 0.0;
	fY		:= MAX(MIN(fBias, fMaxOutput), fMinOutput);
	_fYi	:= 0.0;
	_fbYd(X:= 0.0, T:= 0.0, Y=> );
	RETURN;
END_IF

(* 3. save old variable *)
_fEOld := _fE;

(* 4. set error/deviation input *)
_fE := fSetpoint - fPresentValue;

(* 5. YP-part *)
_fYp := fKp * _fE;

(* 6. YI-part *)
IF (fKi = 0.0) THEN
	_fYi	:= 0.0;
ELSE
	_fYi := _fYi + (fKi * fCtrlCycleTime * _fE);
END_IF
IF (_fYi > fMaxOutput) THEN
	(* limit wind up positive *)
	_fYi := fMaxOutput;
ELSIF (_fYi < fMinOutput) THEN
	(* limit wind up negative *)
	_fYi := fMinOutput;
END_IF

(* 7. YD-part *)
IF (fTp < 0.0) THEN
	fTp := fKd / 10.0;
END_IF
_fYd := fKd * (_fE - _fEOld) / fCtrlCycleTime;
_fbYd(X:= _fYd, T:= fTp, Tcycle:= fCtrlCycleTime, Y=> );

(* 8. Ysum = YP + YI + YD + Bias and output *)
fY := _fYp + _fYi + _fbYd.Y + fBias;
fY := MAX(MIN(fY, fMaxOutput), fMinOutput);

END_FUNCTION_BLOCK

// POUs/Helper/FB_BACnet_PT1
FUNCTION_BLOCK FB_BACnet_PT1
VAR_INPUT
	X : REAL; (* input value *)
	T : REAL; (* damping time [s] *)
	Tcycle : REAL; (* cycle time [s] of task; 0 = use internal measuring *)
END_VAR
VAR_OUTPUT
	Y : REAL; (* damped value *)
END_VAR
VAR
	_sysTime	: GETCPUCOUNTER;
	_Time		: T_LARGE_INTEGER;
	_TimeOld	: T_LARGE_INTEGER;
	_tCycleTime	: REAL;
	_Yold : REAL;
	_FirstScan : BOOL := TRUE;
END_VAR

(* determine cycle time *)
IF Tcycle = 0.0 THEN
	_TimeOld := _Time;
	_sysTime(cpuCntLoDW=> _Time.dwLowPart, cpuCntHiDW=> _Time.dwHighPart);
	_tCycleTime := F_BACnet_SysTimeDiff(In1:=_Time, In2:=_TimeOld);
ELSE
	_tCycleTime := Tcycle;
END_IF

(* exit on wrong cycle time *)
IF _tCycleTime <= 0.0 THEN
	RETURN;
END_IF

(* initialize and check on zero/negative damping time *)
IF (T <= 0.0) OR _FirstScan THEN
	Y := X;
	_Yold := Y;
	_FirstScan := FALSE;
	RETURN;
END_IF

(* remind last result *)
_Yold := Y;

(* calculate result *)
Y := 1 / ((T / _tCycleTime) + 1) * (X - _Yold) + _Yold;

END_FUNCTION_BLOCK

// POUs/Local/Objects/[Base]/FB_BACnet_BasePC
// Pulse Converter Object
{attribute 'enable_dynamic_creation'}
FUNCTION_BLOCK FB_BACnet_BasePC EXTENDS FB_BACnet_EventObject
VAR_INPUT CONSTANT PERSISTENT
	{region 'Variable Parameters'}
		{attribute 'parameterCategory':='Config'}
		fScaleFactor : REAL := 1;	 
				  
		{attribute 'parameterCategory':='Value'}
		fCOVIncrement : REAL := 0.1;
		{attribute 'parameterCategory':='Value'}
		nCovPeriod : UDINT; 	
		{attribute 'parameterCategory':='Value'}
		eUnit : E_BA_Unit := E_BA_Unit.eOther_NoUnits;
			 
		{attribute 'parameterCategory':='EventConfig'}
		bLowLimitEnable : BOOL := FALSE;
		{attribute 'parameterCategory':='EventConfig'}
		fLowLimit : REAL;
		{attribute 'parameterCategory':='EventConfig'}
		bHighLimitEnable : BOOL := FALSE;
		{attribute 'parameterCategory':='EventConfig'}
		fHighLimit : REAL;
		{attribute 'parameterCategory':='EventConfig'}
		fDeadband : REAL := 0.0;
	 
	{endregion}
END_VAR
VAR_OUTPUT
	fPresVal			: REAL;
	nCount				: UDINT;
END_VAR
VAR PERSISTENT
	{region 'Output Parameters'}
		{attribute 'parameterCategory':='Value'}
		fAdjustValue : REAL;
		{attribute 'parameterCategory':='Value'}	
	 	stUpdateTime : ST_BA_DateTime;
		{attribute 'parameterCategory':='Value'}	
		stCountChangeTime : ST_BA_DateTime;
		{attribute 'parameterCategory':='Value'}
		nCountBeforeChange : UDINT;	
	{endregion}
END_VAR

SUPER^();

METHOD PROTECTED OnObjectStateChanged
SUPER^.OnObjectStateChanged();

CASE (tState) OF
	TCOM_STATE.TCOM_STATE_PREOP:
		// SyncHandler:
		RequestSyncHandlers(15, 9);
		
	TCOM_STATE.TCOM_STATE_SAFEOP:
		SyncProperty(E_BACnetPropIdentifier.PropPresentValue, SIZEOF(fPresVal), ADR(fPresVal), 0, eSync_FromSupplement);
		SyncProperty(E_BACnetPropIdentifier.PropCount, SIZEOF(nCount), ADR(nCount), 0, eSync_FromSupplement);
	
	TCOM_STATE.TCOM_STATE_OP:
		SyncProperty(E_BACnetPropIdentifier.PropUnits, SIZEOF(eUnit), ADR(eUnit), 0, eFullSync_InitPLC);
		SyncProperty(E_BACnetPropIdentifier.PropCovIncrement, SIZEOF(fCOVIncrement), ADR(fCOVIncrement), 0, eFullSync_InitPLC);
		SyncProperty(E_BACnetPropIdentifier.PropScaleFactor, SIZEOF(fScaleFactor), ADR(fScaleFactor), 0, eFullSync_InitPLC);
		SyncProperty(E_BACnetPropIdentifier.PropCovPeriod, SIZEOF(nCovPeriod), ADR(nCovPeriod), 0, eFullSync_InitPLC);
			
		SyncPropertyIdx(E_BACnetPropIdentifier.PropLimitEnable, SIZEOF(BOOL), ADR(bHighLimitEnable), E_BACnet_LimitEnableBits.eHighLimit, 0, eFullSync_InitPLC);	
		SyncPropertyIdx(E_BACnetPropIdentifier.PropLimitEnable, SIZEOF(BOOL), ADR(bLowLimitEnable), E_BACnet_LimitEnableBits.eLowLimit, 0, eFullSync_InitPLC);
		SyncProperty(E_BACnetPropIdentifier.PropHighLimit, SIZEOF(fHighLimit), ADR(fHighLimit), 0, eFullSync_InitPLC);
		SyncProperty(E_BACnetPropIdentifier.PropLowLimit, SIZEOF(fLowLimit), ADR(fLowLimit), 0, eFullSync_InitPLC);
		SyncProperty(E_BACnetPropIdentifier.PropDeadband, SIZEOF(fDeadband), ADR(fDeadband), 0, eFullSync_InitPLC);
		
		SyncProperty(E_BACnetPropIdentifier.PropAdjustValue, SIZEOF(REAL), ADR(fAdjustValue), 0, eSync_FromSupplementInitPLC);
	 	SyncProperty(E_BACnetPropIdentifier.PropUpdateTime, SIZEOF(ST_BA_DateTime), ADR(stUpdateTime), 0, eSync_FromSupplementInitPLC);
		SyncProperty(E_BACnetPropIdentifier.PropCountChangeTime, SIZEOF(ST_BA_DateTime), ADR(stCountChangeTime), 0, eSync_FromSupplementInitPLC);
		SyncProperty(E_BACnetPropIdentifier.PropCountBeforeChange, SIZEOF(UDINT), ADR(nCountBeforeChange), 0, eSync_FromSupplementInitPLC);

END_CASE
END_METHOD

METHOD FB_init : BOOL
VAR_INPUT
	bInitRetains : BOOL; // if TRUE, the retain variables are initialized (warm start / cold start)
	bInCopyCode : BOOL;  // if TRUE, the instance afterwards gets moved into the copy code (online change)
END_VAR
eObjectType := E_BACnetObjType.ObjPulseConverter;
END_METHOD

END_FUNCTION_BLOCK

// POUs/Local/Objects/[Base]/FB_BACnet_BaseTLog
FUNCTION_BLOCK ABSTRACT FB_BACnet_BaseTLog EXTENDS FB_BACnet_EventObject
VAR_INPUT CONSTANT PERSISTENT
	{region 'Fixed Parameters'}
		{attribute 'parameterCategory':='Value'}
		nBufferSize : UDINT := BACnet_Param.nLog_BufferEntryCount;
	{endregion}
	{region 'Variable Parameters'}
		{attribute 'parameterCategory':='State'}
		bLogEnable : BOOL;
		
		{attribute 'parameterCategory':='Config'}
		stStartTime : ST_BA_DateTime;
		{attribute 'parameterCategory':='Config'}
		stStopTime : ST_BA_DateTime;
		{attribute 'parameterCategory':='Config'}
		bStopWhenFull : BOOL;
		{attribute 'parameterCategory':='Config'}
		{attribute 'parameterUnit':= '1/100s'}
		nLogInterval : UDINT := 90000;
		{attribute 'parameterCategory':='Config'}
		nNotificationThreshold : UDINT := 50;
		{attribute 'parameterCategory':='Config'}
		eLoggingType : E_BA_LoggingType := E_BA_LoggingType.ePolled;
	{endregion}
END_VAR
VAR_OUTPUT
	nRecCnt							: UDINT;
	nTotRecCnt						: UDINT;
END_VAR
VAR PERSISTENT
	{region 'Output-Properties'}
		nLastNotifyRecord			: UDINT;
		nRecordsSinceNotification	: UDINT;
	{endregion}
END_VAR

SUPER^();

METHOD PROTECTED OnObjectStateChanged
VAR
	_pBufferVal		: PVOID;
	_nBufferSize	: DINT;
END_VAR
SUPER^.OnObjectStateChanged();

CASE (tState) OF
	TCOM_STATE.TCOM_STATE_PREOP:
		// SyncHandler:
		RequestSyncHandlers(11, 8);
		
		// Properties:
		// May limit buffer size to respect array size:
		nBufferSize := MIN(BACnet_Param.nLog_BufferEntryCount, nBufferSize);
		
		WritePropertyUDInt(E_BACnetPropIdentifier.PropBufferSize, nBufferSize);
		
	TCOM_STATE.TCOM_STATE_SAFEOP:
		;

	TCOM_STATE.TCOM_STATE_OP:
		// Synchronize:
		SyncProperty(E_BACnetPropIdentifier.PropLastNotifyRecord, SIZEOF(nLastNotifyRecord), ADR(nLastNotifyRecord), 0, eSync_FromSupplementInitPLC);
		SyncProperty(E_BACnetPropIdentifier.PropRecordsSinceNotification, SIZEOF(nRecordsSinceNotification), ADR(nRecordsSinceNotification), 0, eSync_FromSupplementInitPLC);			
	
		SyncProperty(E_BACnetPropIdentifier.PropTotalRecordCount, SIZEOF(nTotRecCnt), ADR(nTotRecCnt), 0, eSync_FromSupplement);		
		SyncProperty(E_BACnetPropIdentifier.PropRecordCount, SIZEOF(nRecCnt), ADR(nRecCnt), 0, eFullSync_InitPLC);
		SyncProperty(E_BACnetPropIdentifier.PropEnable, SIZEOF(bLogEnable), ADR(bLogEnable), 0, eFullSync_InitPLC);
		SyncProperty(E_BACnetPropIdentifier.PropStartTime, SIZEOF(stStartTime), ADR(stStartTime), 0, eFullSync_InitPLC);
		SyncProperty(E_BACnetPropIdentifier.PropStopTime, SIZEOF(stStopTime), ADR(stStopTime), 0, eFullSync_InitPLC);
		SyncProperty(E_BACnetPropIdentifier.PropStopWhenFull, SIZEOF(bStopWhenFull), ADR(bStopWhenFull), 0, eFullSync_InitPLC);
		SyncProperty(E_BACnetPropIdentifier.PropNotificationThreshold, SIZEOF(nNotificationThreshold), ADR(nNotificationThreshold), 0, eFullSync_InitPLC);
		
		CASE (eObjectType) OF
			E_BACnetObjType.ObjTrendLog,
			E_BACnetObjType.ObjTrendLogMultiple:
				SyncProperty(E_BACnetPropIdentifier.PropLogInterval, SIZEOF(nLogInterval), ADR(nLogInterval), 0, eFullSync_InitPLC);
				SyncProperty(E_BACnetPropIdentifier.PropLoggingType, SIZEOF(eLoggingType), ADR(eLoggingType), 0, eFullSync_InitPLC);
		END_CASE
		
END_CASE
END_METHOD

PROPERTY LastNotifyRecord : UDINT
GET
LastNotifyRecord := nLastNotifyRecord;
END_GET
END_PROPERTY

PROPERTY RecordsSinceNotification : UDINT
GET
RecordsSinceNotification := nRecordsSinceNotification;
END_GET
END_PROPERTY

END_FUNCTION_BLOCK

// POUs/Local/Objects/[Internal]/5P/FB_BACnet_AO_5P
// Analog Output Object
// - Terminal communication
// - 5 Priorities
{attribute 'pin_presentation_order_inputs' := 'bEnSfty,fValSfty,bEnCrit,fValCrit,bEnManLoc,fValManLoc,bEnPgm,fValPgm'}
{attribute 'pin_presentation_order_outputs' := 'fPresVal,eActPrio,bEvent,eRlbty'}
FUNCTION_BLOCK FB_BACnet_AO_5P EXTENDS FB_BACnet_AO
VAR_INPUT
	bEnSfty					: BOOL;
	fValSfty				: REAL;
	bEnCrit					: BOOL;
	fValCrit				: REAL;
	bEnManLoc				: BOOL;
	fValManLoc				: REAL;
END_VAR
VAR_INPUT CONSTANT PERSISTENT
	{region 'Operational Parameters'}
		{attribute 'parameterCategory':='Manual'}
		bEnManualOperator : BOOL;
		{attribute 'parameterCategory':='Manual'}
		fValManualOperator : REAL;
	{endregion}
END_VAR

SUPER^();

METHOD PROTECTED OnObjectStateChanged
SUPER^.OnObjectStateChanged();

CASE (tState) OF
	TCOM_STATE.TCOM_STATE_PREOP:
		// SyncHandler:
		RequestSyncHandlers(4, 4);
		
	TCOM_STATE.TCOM_STATE_SAFEOP:
		SyncPropertyPvPrio(E_BACnetPropIdentifier.PropPresentValue, SIZEOF(fValSfty), ADR(fValSfty), ADR(bEnSfty), BACnet_Param.ePrio_LifeSafety, 0, eFullSync_InitPLC);
		SyncPropertyPvPrio(E_BACnetPropIdentifier.PropPresentValue, SIZEOF(fValCrit), ADR(fValCrit), ADR(bEnCrit), BACnet_Param.ePrio_Critical, 0, eFullSync_InitPLC);
		SyncPropertyPvPrio(E_BACnetPropIdentifier.PropPresentValue, SIZEOF(fValManLoc), ADR(fValManLoc), ADR(bEnManLoc), BACnet_Param.ePrio_ManLocal, 0, eFullSync_InitPLC);
		SyncPropertyPvPrio(E_BACnetPropIdentifier.PropPresentValue, SIZEOF(fValManualOperator), ADR(fValManualOperator), ADR(bEnManualOperator), BACnet_Param.ePrio_ManOperator, 0, eFullSync_InitPLC);
		
	TCOM_STATE.TCOM_STATE_OP:
		;
	
END_CASE
END_METHOD

PROPERTY EnManualOperator : BOOL
GET
EnManualOperator := bEnManualOperator;
END_GET
SET
bEnManualOperator := EnManualOperator;
END_SET
END_PROPERTY

PROPERTY ValManualOperator : REAL
GET
ValManualOperator := fValManualOperator;
END_GET
SET
fValManualOperator := ValManualOperator;
END_SET
END_PROPERTY

END_FUNCTION_BLOCK

// POUs/Local/Objects/FB_BACnet_AO
// Analog Output Object
// - process value
// - 1 Priority
{attribute 'pin_presentation_order_outputs' := 'fPresVal,bEvent,eRlbty'}
{attribute 'enable_dynamic_creation'}
FUNCTION_BLOCK FB_BACnet_AO EXTENDS FB_BACnet_BaseAO
VAR_INPUT	
	eRlbtyPgm 			: E_BA_Reliability;
	bRawOvrrd			: BOOL;					// Raw overridden
END_VAR

IF (bReady) THEN
	// Overridden IO:
	_bOverriddenValue := bRawOvrrd;
END_IF

SUPER^();

METHOD PROTECTED OnObjectStateChanged
SUPER^.OnObjectStateChanged();

CASE (tState) OF
	TCOM_STATE.TCOM_STATE_PREOP:
		// SyncHandler:
		RequestSyncHandlers(0, 2);

	TCOM_STATE.TCOM_STATE_SAFEOP:
		SyncProperty(E_BACnetPropIdentifier.PropReliability, SIZEOF(eRlbtyPgm), ADR(eRlbtyPgm), 0, eSync_ToSupplement);
		
	TCOM_STATE.TCOM_STATE_OP:
		;

END_CASE
END_METHOD

END_FUNCTION_BLOCK

// POUs/Local/Objects/[Internal]/5P/FB_BACnet_AO_IO5P
// Analog Output Object
// - Terminal communication
// - 5 Priorities
{attribute 'pin_presentation_order_inputs' := 'bEnSfty,fValSfty,bEnCrit,fValCrit,bEnManLoc,fValManLoc,bEnPgm,fValPgm'}
{attribute 'pin_presentation_order_outputs' := 'fPresVal,eActPrio,bEvent,eRlbty'}
FUNCTION_BLOCK FB_BACnet_AO_IO5P EXTENDS FB_BACnet_AO_IO
VAR_INPUT
	bEnSfty					: BOOL;
	fValSfty				: REAL;
	bEnCrit					: BOOL;
	fValCrit				: REAL;
	bEnManLoc				: BOOL;
	fValManLoc				: REAL;
END_VAR
VAR_INPUT CONSTANT PERSISTENT
	{region 'Operational Parameters'}
		{attribute 'parameterCategory':='Manual'}
		bEnManualOperator : BOOL;
		{attribute 'parameterCategory':='Manual'}
		fValManualOperator : REAL;
	{endregion}
END_VAR

SUPER^();

METHOD PROTECTED OnObjectStateChanged
SUPER^.OnObjectStateChanged();

CASE (tState) OF
	TCOM_STATE.TCOM_STATE_PREOP:
		// SyncHandler:
		RequestSyncHandlers(4, 4);
		
	TCOM_STATE.TCOM_STATE_SAFEOP:
		SyncPropertyPvPrio(E_BACnetPropIdentifier.PropPresentValue, SIZEOF(fValSfty), ADR(fValSfty), ADR(bEnSfty), BACnet_Param.ePrio_LifeSafety, 0, eFullSync_InitPLC);
		SyncPropertyPvPrio(E_BACnetPropIdentifier.PropPresentValue, SIZEOF(fValCrit), ADR(fValCrit), ADR(bEnCrit), BACnet_Param.ePrio_Critical, 0, eFullSync_InitPLC);
		SyncPropertyPvPrio(E_BACnetPropIdentifier.PropPresentValue, SIZEOF(fValManLoc), ADR(fValManLoc), ADR(bEnManLoc), BACnet_Param.ePrio_ManLocal, 0, eFullSync_InitPLC);
		SyncPropertyPvPrio(E_BACnetPropIdentifier.PropPresentValue, SIZEOF(fValManualOperator), ADR(fValManualOperator), ADR(bEnManualOperator), BACnet_Param.ePrio_ManOperator, 0, eFullSync_InitPLC);
		
	TCOM_STATE.TCOM_STATE_OP:
		;
	
END_CASE
END_METHOD

PROPERTY EnManualOperator : BOOL
GET
EnManualOperator := bEnManualOperator;
END_GET
SET
bEnManualOperator := EnManualOperator;
END_SET
END_PROPERTY

PROPERTY ValManualOperator : REAL
GET
ValManualOperator := fValManualOperator;
END_GET
SET
fValManualOperator := ValManualOperator;
END_SET
END_PROPERTY

END_FUNCTION_BLOCK

// POUs/Local/Objects/FB_BACnet_AO_IO
// Analog Output Object
// - Terminal communication
// - 1 Priority
{attribute 'pin_presentation_order_outputs' := 'fPresVal,bEvent,eRlbty'}
FUNCTION_BLOCK FB_BACnet_AO_IO EXTENDS FB_BACnet_BaseAO
VAR_INPUT CONSTANT PERSISTENT
	{region 'Fixed Parameters'}
		{attribute 'parameterCategory':='Hardware'}
		nIoBusNr : BYTE := 16#FF;
	{endregion}
	{region 'Variable Parameters'}
		{attribute 'parameterCategory':='Config'}
		eOverriddenPolarity : E_BA_Polarity := E_BA_Polarity.eNormal;
	{endregion}
END_VAR
VAR
	{region 'Raw I/O'}
		bRawOvrrd			AT %I*	: BOOL;				// Raw overridden (Optional)
		nRawState			AT %I*	: USINT;			// Raw state (Optional, only used to determine overridden state)
		nRawValue			AT %Q*	: INT;				// Raw value
	{endregion}
	{region 'Hardware'}
		_bIsOverriddenMapped		: BOOL;				// Indication to mapped hardware for overridden IO value
		_bIsStateMapped				: BOOL;				// Indication to mapped hardware for state
	{endregion}
END_VAR

IF (bReady) THEN
	// Overridden IO Value:
	IF (_bIsOverriddenMapped) THEN
		_bOverriddenValue := (bRawOvrrd = (eOverriddenPolarity=E_BA_Polarity.eNormal));
	ELSIF (_bIsStateMapped) THEN
		_bOverriddenValue := ((nRawState=0) = (eOverriddenPolarity=E_BA_Polarity.eNormal));
	ELSE
		_bOverriddenValue := FALSE;
	END_IF
END_IF

SUPER^();

METHOD PROTECTED OnObjectStateChanged
SUPER^.OnObjectStateChanged();

CASE (tState) OF
	TCOM_STATE.TCOM_STATE_PREOP:
		// SyncHandler:
		RequestSyncHandlers(1, 0);

		IF (nIoBusNr <> 16#FF) THEN
			WritePropertyByte(E_BACnetPropIdentifier.PropIoBusNr, nIoBusNr);
		END_IF
		
	TCOM_STATE.TCOM_STATE_SAFEOP:
		SyncProperty(E_BACnetPropIdentifier.PropRawIoAnalogValueINT, SIZEOF(nRawValue), ADR(nRawValue), 0, eSync_FromSupplement);
		
	TCOM_STATE.TCOM_STATE_OP:
		// Check mapping of state:
		_bIsStateMapped := (F_GetMappingStatus(ADR(nRawState), SIZEOF(nRawState)) <> EPlcMappingStatus.MS_Unmapped);
		// Check mapping of overridden IO:
		_bIsOverriddenMapped := (F_GetMappingStatus(ADR(bRawOvrrd), SIZEOF(bRawOvrrd)) <> EPlcMappingStatus.MS_Unmapped);
		
END_CASE
END_METHOD

END_FUNCTION_BLOCK

// POUs/Local/Objects/[Internal]/5P/FB_BACnet_BO_5P
// Binary Output Object
// - Terminal communication
// - 5 Priorities
{attribute 'pin_presentation_order_inputs' := 'bEnSfty,bValSfty,bEnCrit,bValCrit,bEnManLoc,bValManLoc,bEnPgm,bValPgm'}
{attribute 'pin_presentation_order_outputs' := 'bPresVal,eActPrio,bEvent,eRlbty'}
FUNCTION_BLOCK FB_BACnet_BO_5P EXTENDS FB_BACnet_BO
VAR_INPUT
	bEnSfty					: BOOL;
	bValSfty				: BOOL;
	bEnCrit					: BOOL;
	bValCrit				: BOOL;
	bEnManLoc				: BOOL;
	bValManLoc				: BOOL;
END_VAR
VAR_INPUT CONSTANT PERSISTENT
	{region 'Operational Parameters'}
		{attribute 'parameterCategory':='Manual'}
		bEnManualOperator : BOOL;
		{attribute 'parameterCategory':='Manual'}
		bValManualOperator : BOOL;
	{endregion}
END_VAR

SUPER^();

METHOD PROTECTED OnObjectStateChanged
SUPER^.OnObjectStateChanged();

CASE (tState) OF
	TCOM_STATE.TCOM_STATE_PREOP:
		// SyncHandler:
		RequestSyncHandlers(4, 4);
		
	TCOM_STATE.TCOM_STATE_SAFEOP:
		SyncPropertyPvPrio(E_BACnetPropIdentifier.PropPresentValue, SIZEOF(bValSfty), ADR(bValSfty), ADR(bEnSfty), BACnet_Param.ePrio_LifeSafety, 0, eFullSync_InitPLC);
		SyncPropertyPvPrio(E_BACnetPropIdentifier.PropPresentValue, SIZEOF(bValCrit), ADR(bValCrit), ADR(bEnCrit), BACnet_Param.ePrio_Critical, 0, eFullSync_InitPLC);
		SyncPropertyPvPrio(E_BACnetPropIdentifier.PropPresentValue, SIZEOF(bValManLoc), ADR(bValManLoc), ADR(bEnManLoc), BACnet_Param.ePrio_ManLocal, 0, eFullSync_InitPLC);
		SyncPropertyPvPrio(E_BACnetPropIdentifier.PropPresentValue, SIZEOF(bValManualOperator), ADR(bValManualOperator), ADR(bEnManualOperator), BACnet_Param.ePrio_ManOperator, 0, eFullSync_InitPLC);
		
	TCOM_STATE.TCOM_STATE_OP:
		;
		
END_CASE
END_METHOD

PROPERTY EnManualOperator : BOOL
GET
EnManualOperator := bEnManualOperator;
END_GET
SET
bEnManualOperator := EnManualOperator;
END_SET
END_PROPERTY

PROPERTY ValManualOperator : BOOL
GET
ValManualOperator := bValManualOperator;
END_GET
SET
bValManualOperator := ValManualOperator;
END_SET
END_PROPERTY

END_FUNCTION_BLOCK

// POUs/Local/Objects/FB_BACnet_BO
// Binary Output Object
// - process value
// - 1 Priority
{attribute 'pin_presentation_order_outputs' := 'fPresVal,bEvent,eRlbty'}
{attribute 'enable_dynamic_creation'}
FUNCTION_BLOCK FB_BACnet_BO EXTENDS FB_BACnet_BaseBO
VAR_INPUT
	bRawOvrrd					: BOOL;				// Raw overridden
	bEnFdbck					: BOOL;				// Enable of writing to Feedback Value (optional)
	bRawValFdbck				: BOOL;				// Raw feedback Value
	eRlbtyPgm 					: E_BA_Reliability;
END_VAR

IF (bReady) THEN
	// Feedback Value:
	_bFeedbackValue := SEL(bEnFdbck, bPresVal, bRawValFdbck);
END_IF

SUPER^();

METHOD PROTECTED OnObjectStateChanged
SUPER^.OnObjectStateChanged();

CASE (tState) OF
	TCOM_STATE.TCOM_STATE_PREOP:
		// SyncHandler:
		RequestSyncHandlers(1, 1);

	TCOM_STATE.TCOM_STATE_SAFEOP:
		SyncProperty(E_BACnetPropIdentifier.PropRawIoStateOverride, SIZEOF(bRawOvrrd), ADR(bRawOvrrd), 0, eSync_ToSupplement);
		SyncProperty(E_BACnetPropIdentifier.PropReliability, SIZEOF(eRlbtyPgm), ADR(eRlbtyPgm), 0, eSync_ToSupplement);
		
	TCOM_STATE.TCOM_STATE_OP:
		;

END_CASE
END_METHOD

END_FUNCTION_BLOCK

// POUs/Local/Objects/[Internal]/5P/FB_BACnet_BO_IO5P
// Binary Output Object
// - Terminal communication
// - 5 Priorities
{attribute 'pin_presentation_order_inputs' := 'bEnSfty,bValSfty,bEnCrit,bValCrit,bEnManLoc,bValManLoc,bEnPgm,bValPgm'}
{attribute 'pin_presentation_order_outputs' := 'bPresVal,eActPrio,bEvent,eRlbty'}
FUNCTION_BLOCK FB_BACnet_BO_IO5P EXTENDS FB_BACnet_BO_IO
VAR_INPUT
	bEnSfty					: BOOL;
	bValSfty				: BOOL;
	bEnCrit					: BOOL;
	bValCrit				: BOOL;
	bEnManLoc				: BOOL;
	bValManLoc				: BOOL;
END_VAR
VAR_INPUT CONSTANT PERSISTENT
	{region 'Operational Parameters'}
		{attribute 'parameterCategory':='Manual'}
		bEnManualOperator : BOOL;
		{attribute 'parameterCategory':='Manual'}
		bValManualOperator : BOOL;
	{endregion}
END_VAR

SUPER^();

METHOD PROTECTED OnObjectStateChanged
SUPER^.OnObjectStateChanged();

CASE (tState) OF
	TCOM_STATE.TCOM_STATE_PREOP:
		// SyncHandler:
		RequestSyncHandlers(4, 4);
		
	TCOM_STATE.TCOM_STATE_SAFEOP:
		SyncPropertyPvPrio(E_BACnetPropIdentifier.PropPresentValue, SIZEOF(bValSfty), ADR(bValSfty), ADR(bEnSfty), BACnet_Param.ePrio_LifeSafety, 0, eFullSync_InitPLC);
		SyncPropertyPvPrio(E_BACnetPropIdentifier.PropPresentValue, SIZEOF(bValCrit), ADR(bValCrit), ADR(bEnCrit), BACnet_Param.ePrio_Critical, 0, eFullSync_InitPLC);
		SyncPropertyPvPrio(E_BACnetPropIdentifier.PropPresentValue, SIZEOF(bValManLoc), ADR(bValManLoc), ADR(bEnManLoc), BACnet_Param.ePrio_ManLocal, 0, eFullSync_InitPLC);
		SyncPropertyPvPrio(E_BACnetPropIdentifier.PropPresentValue, SIZEOF(bValManualOperator), ADR(bValManualOperator), ADR(bEnManualOperator), BACnet_Param.ePrio_ManOperator, 0, eFullSync_InitPLC);
		
	TCOM_STATE.TCOM_STATE_OP:
		;
		
END_CASE
END_METHOD

PROPERTY EnManualOperator : BOOL
GET
EnManualOperator := bEnManualOperator;
END_GET
SET
bEnManualOperator := EnManualOperator;
END_SET
END_PROPERTY

PROPERTY ValManualOperator : BOOL
GET
ValManualOperator := bValManualOperator;
END_GET
SET
bValManualOperator := ValManualOperator;
END_SET
END_PROPERTY

END_FUNCTION_BLOCK

// POUs/Local/Objects/FB_BACnet_BO_IO
// Binary Output Object
// - Terminal communication
// - 1 Priority
{attribute 'pin_presentation_order_outputs' := 'fPresVal,bEvent,eRlbty'}
FUNCTION_BLOCK FB_BACnet_BO_IO EXTENDS FB_BACnet_BaseBO
VAR_INPUT CONSTANT PERSISTENT
	{region 'Fixed Parameters'}
		{attribute 'parameterCategory':='Hardware'}
		nIoBusNr : BYTE := 16#FF;
	{endregion}
	{region 'Variable Parameters'}
		{attribute 'parameterCategory':='Config'}
		eFeedbackPolarity : E_BA_Polarity := E_BA_Polarity.eNormal;
		{attribute 'parameterCategory':='Config'}
		eOverriddenPolarity : E_BA_Polarity := E_BA_Polarity.eNormal;
	{endregion}
END_VAR
VAR
	{region 'Raw I/O'}
		bRawOverridden		AT %I*	: BOOL;				// Raw overridden (Optional)
		bRawValFeedback		AT %I*	: BOOL;				// Raw feedback Value (Optional)
		bRawValue			AT %Q*	: BOOL;				// Raw value
	{endregion}
	{region 'Hardware'}
		_bIsFeedbackMapped			: BOOL;				// Indication to mapped hardware for feedback value
		_bIsOverriddenMapped		: BOOL;				// Indication to mapped hardware for overridden IO value
	{endregion}
	{region 'Internal'}
		_bOverriddenValue			: BOOL;
	{endregion}
END_VAR
VAR_STAT 
	{region 'Temporary'}
		{attribute 'hide'}
		_bEnFeedback				: BOOL;
	{endregion}
END_VAR

IF (bReady) THEN
	// Overridden IO Value:
	_bOverriddenValue := SEL(_bIsOverriddenMapped, FALSE, (bRawOverridden = (eOverriddenPolarity=E_BA_Polarity.eNormal)));
	
	// Feedback Value:
	_bEnFeedback := SEL(_bIsFeedbackMapped, FALSE, NOT _bOverriddenValue);
	_bFeedbackValue := SEL(_bEnFeedback, bPresVal, (bRawValFeedback = (eFeedbackPolarity=E_BA_Polarity.eNormal)));
END_IF

SUPER^();

METHOD PROTECTED OnObjectStateChanged
SUPER^.OnObjectStateChanged();

CASE (tState) OF
	TCOM_STATE.TCOM_STATE_PREOP:
		// SyncHandler:
		RequestSyncHandlers(1, 1);

		IF (nIoBusNr <> 16#FF) THEN
			WritePropertyByte(E_BACnetPropIdentifier.PropIoBusNr, nIoBusNr);
		END_IF
		
	TCOM_STATE.TCOM_STATE_SAFEOP:
		SyncProperty(E_BACnetPropIdentifier.PropRawIoBinaryValueBOOL, SIZEOF(bRawValue), ADR(bRawValue), 0, eSync_FromSupplement);
		SyncProperty(E_BACnetPropIdentifier.PropRawIoStateOverride, SIZEOF(_bOverriddenValue), ADR(_bOverriddenValue), 0, eSync_ToSupplement);
		
	TCOM_STATE.TCOM_STATE_OP:
		
		// Check mapping of feedback:
		_bIsFeedbackMapped := (F_GetMappingStatus(ADR(bRawValFeedback), SIZEOF(bRawValFeedback)) <> EPlcMappingStatus.MS_Unmapped);
		// Check mapping of overridden IO:
		_bIsOverriddenMapped := (F_GetMappingStatus(ADR(bRawOverridden), SIZEOF(bRawOverridden)) <> EPlcMappingStatus.MS_Unmapped);
		
END_CASE
END_METHOD

END_FUNCTION_BLOCK

// POUs/Local/Objects/[Internal]/5P/FB_BACnet_MO_5P
// Multistate Output Object
// - Terminal communication
// - 5 Priorities
{attribute 'pin_presentation_order_inputs' := 'bEnSfty,nValSfty,bEnCrit,nValCrit,bEnManLoc,nValManLoc,bEnPgm,nValPgm'}
{attribute 'pin_presentation_order_outputs' := 'nPresVal,eActPrio,bEvent,eRlbty'}
FUNCTION_BLOCK FB_BACnet_MO_5P EXTENDS FB_BACnet_MO
VAR_INPUT
	bEnSfty					: BOOL;
	nValSfty				: UDINT		:= 1;
	bEnCrit					: BOOL;
	nValCrit				: UDINT		:= 1;
	bEnManLoc				: BOOL;
	nValManLoc				: UDINT		:= 1;
END_VAR
VAR_INPUT CONSTANT PERSISTENT
	{region 'Operational Parameters'}
		{attribute 'parameterCategory':='Manual'}
		bEnManualOperator : BOOL;
		{attribute 'parameterCategory':='Manual'}
		nValManualOperator : UDINT := 1;
	{endregion}
END_VAR

SUPER^();

METHOD PROTECTED OnObjectStateChanged
SUPER^.OnObjectStateChanged();

CASE (tState) OF
	TCOM_STATE.TCOM_STATE_PREOP:
		// SyncHandler:
		RequestSyncHandlers(4, 4);
		
	TCOM_STATE.TCOM_STATE_SAFEOP:
		SyncPropertyPvPrio(E_BACnetPropIdentifier.PropPresentValue, SIZEOF(nValSfty), ADR(nValSfty), ADR(bEnSfty), BACnet_Param.ePrio_LifeSafety, 0, eFullSync_InitPLC);
		SyncPropertyPvPrio(E_BACnetPropIdentifier.PropPresentValue, SIZEOF(nValCrit), ADR(nValCrit), ADR(bEnCrit), BACnet_Param.ePrio_Critical, 0, eFullSync_InitPLC);
		SyncPropertyPvPrio(E_BACnetPropIdentifier.PropPresentValue, SIZEOF(nValManLoc), ADR(nValManLoc), ADR(bEnManLoc), BACnet_Param.ePrio_ManLocal, 0, eFullSync_InitPLC);
		SyncPropertyPvPrio(E_BACnetPropIdentifier.PropPresentValue, SIZEOF(nValManualOperator), ADR(nValManualOperator), ADR(bEnManualOperator), BACnet_Param.ePrio_ManOperator, 0, eFullSync_InitPLC);
		
	TCOM_STATE.TCOM_STATE_OP:
		;
		
END_CASE
END_METHOD

PROPERTY EnManualOperator : BOOL
GET
EnManualOperator := bEnManualOperator;
END_GET
SET
bEnManualOperator := EnManualOperator;
END_SET
END_PROPERTY

PROPERTY ValManualOperator : UDINT
GET
ValManualOperator := nValManualOperator;
END_GET
SET
nValManualOperator := ValManualOperator;
END_SET
END_PROPERTY

END_FUNCTION_BLOCK

// POUs/Local/Objects/FB_BACnet_MO
// Multistate Output Object
// - process value
// - 1 Priority
{attribute 'pin_presentation_order_outputs' := 'fPresVal,bEvent,eRlbty'}
{attribute 'enable_dynamic_creation'}
FUNCTION_BLOCK FB_BACnet_MO EXTENDS FB_BACnet_BaseMO
VAR_INPUT
	bRawOvrrd					: BOOL;				// Raw overridden
	bEnFeedback					: BOOL;				// Enable of writing to Feedback Value (optional)
	nRawValFeedback				: UDINT;			// Raw feedback Value
	eRlbtyPgm 					: E_BA_Reliability;
END_VAR

IF (bReady) THEN
	// Feedback Value:
	_nFeedbackValue := MAX(1, SEL(bEnFeedback, nPresVal, nRawValFeedback));
END_IF

SUPER^();

METHOD PROTECTED OnObjectStateChanged
SUPER^.OnObjectStateChanged();

CASE (tState) OF
	TCOM_STATE.TCOM_STATE_PREOP:
		// SyncHandler:
		RequestSyncHandlers(0, 1);

	TCOM_STATE.TCOM_STATE_SAFEOP:
		SyncProperty(E_BACnetPropIdentifier.PropRawIoStateOverride, SIZEOF(bRawOvrrd), ADR(bRawOvrrd), 0, eSync_ToSupplement);
		SyncProperty(E_BACnetPropIdentifier.PropReliability, SIZEOF(eRlbtyPgm), ADR(eRlbtyPgm), 0, eSync_ToSupplement);
		
	TCOM_STATE.TCOM_STATE_OP:
		;

END_CASE
END_METHOD

END_FUNCTION_BLOCK

// POUs/Local/Objects/[Internal]/5P/FB_BACnet_MO_IO5P
// Multistate Output Object
// - Terminal communication
// - 5 Priorities
{attribute 'pin_presentation_order_inputs' := 'bEnSfty,nValSfty,bEnCrit,nValCrit,bEnManLoc,nValManLoc,bEnPgm,nValPgm'}
{attribute 'pin_presentation_order_outputs' := 'nPresVal,eActPrio,bEvent,eRlbty'}
FUNCTION_BLOCK FB_BACnet_MO_IO5P EXTENDS FB_BACnet_MO_IO
VAR_INPUT
	bEnSfty					: BOOL;
	nValSfty				: UDINT		:= 1;
	bEnCrit					: BOOL;
	nValCrit				: UDINT		:= 1;
	bEnManLoc				: BOOL;
	nValManLoc				: UDINT		:= 1;
END_VAR
VAR_INPUT CONSTANT PERSISTENT
	{region 'Operational Parameters'}
		{attribute 'parameterCategory':='Manual'}
		bEnManualOperator : BOOL;
		{attribute 'parameterCategory':='Manual'}
		nValManualOperator : UDINT := 1;
	{endregion}
END_VAR

SUPER^();

METHOD PROTECTED OnObjectStateChanged
SUPER^.OnObjectStateChanged();

CASE (tState) OF
	TCOM_STATE.TCOM_STATE_PREOP:
		// SyncHandler:
		RequestSyncHandlers(4, 4);
		
	TCOM_STATE.TCOM_STATE_SAFEOP:
		SyncPropertyPvPrio(E_BACnetPropIdentifier.PropPresentValue, SIZEOF(nValSfty), ADR(nValSfty), ADR(bEnSfty), BACnet_Param.ePrio_LifeSafety, 0, eFullSync_InitPLC);
		SyncPropertyPvPrio(E_BACnetPropIdentifier.PropPresentValue, SIZEOF(nValCrit), ADR(nValCrit), ADR(bEnCrit), BACnet_Param.ePrio_Critical, 0, eFullSync_InitPLC);
		SyncPropertyPvPrio(E_BACnetPropIdentifier.PropPresentValue, SIZEOF(nValManLoc), ADR(nValManLoc), ADR(bEnManLoc), BACnet_Param.ePrio_ManLocal, 0, eFullSync_InitPLC);
		SyncPropertyPvPrio(E_BACnetPropIdentifier.PropPresentValue, SIZEOF(nValManualOperator), ADR(nValManualOperator), ADR(bEnManualOperator), BACnet_Param.ePrio_ManOperator, 0, eFullSync_InitPLC);
		
	TCOM_STATE.TCOM_STATE_OP:
		;
		
END_CASE
END_METHOD

PROPERTY EnManualOperator : BOOL
GET
EnManualOperator := bEnManualOperator;
END_GET
SET
bEnManualOperator := EnManualOperator;
END_SET
END_PROPERTY

PROPERTY ValManualOperator : UDINT
GET
ValManualOperator := nValManualOperator;
END_GET
SET
nValManualOperator := ValManualOperator;
END_SET
END_PROPERTY

END_FUNCTION_BLOCK

// POUs/Local/Objects/FB_BACnet_MO_IO
// Multistate Output Object
// - Terminal communication
// - 1 Priority
{attribute 'pin_presentation_order_outputs' := 'fPresVal,bEvent,eRlbty'}
FUNCTION_BLOCK FB_BACnet_MO_IO EXTENDS FB_BACnet_BaseMO
VAR_INPUT CONSTANT PERSISTENT
	{region 'Variable Parameters'}
		{attribute 'parameterCategory':='Config'}
		eMappingMode : E_BA_ByteMappingMode := E_BA_ByteMappingMode.eIndex1N;
		{attribute 'parameterCategory':='Config'}
		eFeedbackMappingMode : E_BA_ByteMappingMode := E_BA_ByteMappingMode.eIndex1N;
	{endregion}
END_VAR
VAR
	{region 'Raw I/O'}
		bRawOverridden		AT %I*	: BOOL;				// Raw overridden (Optional)
		bRawValFeedback		AT %I*	: ST_BA_Byte;		// Bus terminal feedback Value (Optional)
		bRawValue			AT %Q*	: ST_BA_Byte;		// Bus terminal value
	{endregion}
	{region 'Hardware'}
		_bIsFeedbackMapped			: BOOL;				// Indication to mapped hardware for feedback value
	{endregion}
	{region 'Internal'}
		nLastPresentValue			: UDINT;
	{endregion}
END_VAR

IF (bReady) THEN
	// Feedback Value:
	IF (_bIsFeedbackMapped) THEN
		F_BA_MapUDIFromRawByte(_nFeedbackValue, ADR(bRawValFeedback), eFeedbackMappingMode, nRelinquishDefault);
	ELSE
		_nFeedbackValue := nPresVal;
	END_IF
	
	// Trigger change of value:
	IF (nPresVal <> nLastPresentValue) THEN
		nLastPresentValue := nPresVal;
		F_BA_MapUDIToRawByte(nPresVal, ADR(bRawValue), eMappingMode, nRelinquishDefault);
	END_IF
ELSE
	nPresVal := nRelinquishDefault;
	
	// Set last value to a different value compared to actual raw value (So a COV is triggered when current instance becomes ready):
	nLastPresentValue := (nLastPresentValue+1);
END_IF

SUPER^();

METHOD PROTECTED OnObjectStateChanged
SUPER^.OnObjectStateChanged();

CASE (tState) OF
	TCOM_STATE.TCOM_STATE_PREOP:
		// SyncHandler:
		RequestSyncHandlers(0, 1);

	TCOM_STATE.TCOM_STATE_SAFEOP:
		SyncProperty(E_BACnetPropIdentifier.PropRawIoStateOverride, SIZEOF(bRawOverridden), ADR(bRawOverridden), 0, eSync_ToSupplement);
		
	TCOM_STATE.TCOM_STATE_OP:
		// Check mapping of feedback:
		_bIsFeedbackMapped := (F_GetMappingStatus(ADR(bRawValFeedback), SIZEOF(bRawValFeedback)) <> EPlcMappingStatus.MS_Unmapped);
		
END_CASE
END_METHOD

END_FUNCTION_BLOCK

// POUs/Local/Objects/[Internal]/Property/Buffer/[Archiv]/FB_BACnet_WeeklyScheduleBuffer
FUNCTION_BLOCK INTERNAL FB_BACnet_WeeklyScheduleBuffer EXTENDS FB_BACnet_BaseListBuffer

SUPER^();

METHOD ResetValue
VAR
	_nDay : INT;
END_VAR
SUPER^.ResetValue();

// Write empty weekday-array to buffer:
FOR _nDay := E_BA_Weekday.First TO E_BA_Weekday.Last DO
	MemSetULINT(16#0000000080000008, nUsedSize);
	MemSetULINT(16#0000000000000000, nUsedSize);
END_FOR

(*
FOR iDayTmp := iWeekdayFirst TO iWeekdayLast DO
	MemSetULINT(16#0000000080000020, nUsedSize);
	MemSetULINT(16#0000000000000000, nUsedSize);
	MemSetULINT(16#0000000000000000, nUsedSize);
	MemSetULINT(16#0000000000000000, nUsedSize);
	MemSetULINT(16#0000000000000000, nUsedSize);
END_FOR
*)
END_METHOD

METHOD FB_init : BOOL
VAR_INPUT
	bInitRetains : BOOL; // if TRUE, the retain variables are initialized (warm start / cold start)
	bInCopyCode : BOOL;  // if TRUE, the instance afterwards gets moved into the copy code (online change)
END_VAR
ePropertyID := E_BACnetPropIdentifier.PropWeeklySchedule;
END_METHOD

END_FUNCTION_BLOCK

// POUs/Local/Objects/[Internal]/Property/Buffer/Base/FB_BACnet_BaseListBuffer
FUNCTION_BLOCK INTERNAL FB_BACnet_BaseListBuffer EXTENDS FB_BACnet_BasePropertyBuffer
VAR PERSISTENT
	aBuffer : ARRAY[1 .. nBACnet_BufferSize] OF BYTE;
END_VAR
VAR CONSTANT
	{attribute 'hide'}
	{attribute 'parameterUnit':= 'byte'}
	nBACnet_BufferSize	: UINT	:= 8192;
END_VAR

SUPER^();

METHOD PROTECTED ValidateInst : BOOL
nBufferSize := SIZEOF(aBuffer);
pBufferValue := ADR(aBuffer);

ValidateInst := SUPER^.ValidateInst();
END_METHOD

END_FUNCTION_BLOCK

// POUs/Local/Objects/[Internal]/Property/Buffer/Base/FB_BACnet_BasePropertyBuffer
FUNCTION_BLOCK INTERNAL FB_BACnet_BasePropertyBuffer
VAR_OUTPUT
	ePropertyID : E_BACnetPropIdentifier := E_BACnetPropIdentifier.PropInvalid;		// ID of referred property
	bChangeTrig : BOOL;												// Change trigger
	nChanges : UINT;												// Changes counter
	bReady : BOOL;												// Synchronization of referred property successfully initialized
END_VAR
VAR PERSISTENT
	nUsedSize : UDINT;
END_VAR
VAR
	// Init via instance-declaration:
	iRefObject : I_BACnet_Object;
	
	// Init via SubClass:
	tSyncState : TCOM_STATE := TCOM_STATE.TCOM_STATE_OP;						// Object-state to init synchronization of referred property
END_VAR
VAR_STAT
	// Use "ValidateInst()" to ensure data to be valid: 
	{attribute 'hide'}
	fbRefObject : POINTER TO FB_BACnet_Object;
	{attribute 'hide'}
	nBufferSize : UDINT;
	{attribute 'hide'}
	pBufferValue : PVOID;
END_VAR
(*
VAR
	// [DEBUG]:
	eDebugCommand : (eNone:=1, eReadBuffer:=2, eWriteBuffer:=3, eResetBuffer:=4, ePrintBuffer:=5) UDINT := 1;
	sDebugHexBuffer : T_MaxString;
END_VAR
*)

IF (bChangeTrig) THEN
	bChangeTrig := FALSE;
	nChanges := (nChanges+1);
	
	IF (ValidateInst()) THEN
		// Refresh property value:
		ReadValue();
	END_IF
END_IF

(*
// [DEBUG]:
IF (eDebugCommand <> eNone) THEN
	IF (ValidateInst()) THEN
		CASE (eDebugCommand) OF
			eReadBuffer:
				ReadValue();
			eWriteBuffer:
				WriteValue();
			eResetBuffer:
				ResetValue();
			ePrintBuffer:
				sDebugHexBuffer := DATA_TO_HEXSTR(pData:=pBufferValue, cbData:=TO_UDINT(nUsedSize), FALSE);
		END_CASE
	END_IF
	eDebugCommand := eNone;
END_IF
*)

// Write a (any type) value to the memory buffer. 
// > Ensure to point to valid memory buffer via "ValidateInst()"!
METHOD PROTECTED MemSet : BOOL
VAR_INPUT
	xValue : ANY;
END_VAR
VAR_IN_OUT
	nOffset : UDINT;
END_VAR
VAR
	_nSizeTmp : UDINT;
END_VAR
_nSizeTmp := TO_UDINT(xValue.diSize);

IF (pBufferValue = 0) THEN
	F_BA_LogMessage(ADSLOG_MSGTYPE_ERROR, 'MS02', 'PropertyBuffer.MemSet: Uninitialized buffer!');
ELSIF ((_nSizeTmp+nOffset) > nBufferSize) THEN
	F_BA_LogMessage(ADSLOG_MSGTYPE_ERROR, 'MS04', 'PropertyBuffer.MemSet: Buffer size exceeded!');
ELSE
	MEMCPY((pBufferValue+nOffset), xValue.pValue, _nSizeTmp);
	nOffset := (nOffset+_nSizeTmp);
	
	MemSet := TRUE;
END_IF
END_METHOD

// Write a 1Byte-value to the memory buffer. 
METHOD PROTECTED MemSetBYTE : BOOL
VAR_INPUT
	nValue : BYTE;
END_VAR
VAR_IN_OUT
	nOffset : UDINT;
END_VAR
MemSetBYTE := MemSet(nValue, nOffset);
END_METHOD

// Write a 4Byte-value to the memory buffer. 
METHOD PROTECTED MemSetUDINT : BOOL
VAR_INPUT
	nValue : UDINT;
END_VAR
VAR_IN_OUT
	nOffset : UDINT;
END_VAR
MemSetUDINT := MemSet(nValue, nOffset);
END_METHOD

// Write a 2Byte-value to the memory buffer. 
METHOD PROTECTED MemSetUINT : BOOL
VAR_INPUT
	nValue : UINT;
END_VAR
VAR_IN_OUT
	nOffset : UDINT;
END_VAR
MemSetUINT := MemSet(nValue, nOffset);
END_METHOD

// Write a 8Byte-value to the memory buffer. 
METHOD PROTECTED MemSetULINT : BOOL
VAR_INPUT
	nValue : ULINT;
END_VAR
VAR_IN_OUT
	nOffset : UDINT;
END_VAR
MemSetULINT := MemSet(nValue, nOffset);
END_METHOD

METHOD PROTECTED ReadValue : HRESULT
nUsedSize := nBufferSize;
ReadValue := fbRefObject^.ReadProperty(ePropertyID, pBufferValue, ADR(nUsedSize));
END_METHOD

METHOD PROTECTED ValidateInst : BOOL
IF (iRefObject = 0) THEN
	F_BA_LogMessage(ADSLOG_MSGTYPE_ERROR, 'GB3', 'PropertyBuffer: Unreferred object!');
	
ELSIF (NOT __QUERYPOINTER(iRefObject, fbRefObject)) OR (fbRefObject = 0) THEN
	F_BA_LogMessage(ADSLOG_MSGTYPE_ERROR, 'GB6', 'PropertyBuffer: Invalid referred object!');
	
ELSIF (nBufferSize = 0) OR (pBufferValue = 0) THEN
	F_BA_LogMessage1(ADSLOG_MSGTYPE_ERROR, 'GB8', 'PropertyBuffer: Unimplemented buffer of property "%d"!', F_INT(ePropertyID));

ELSE
	ValidateInst := TRUE;
END_IF
END_METHOD

METHOD PROTECTED WriteValue : HRESULT
WriteValue := fbRefObject^.WriteProperty(ePropertyID, pBufferValue, TO_DINT(nUsedSize));
END_METHOD

METHOD OnObjectStateChanged
VAR_INPUT
	tState : TCOM_STATE;
END_VAR
VAR
	eSyncMode : E_BA_FullSyncMode := eFullSync_InitPLC;
END_VAR
IF (tState = tSyncState) THEN
	IF (ePropertyID = E_BACnetPropIdentifier.PropInvalid) THEN
		F_BA_LogMessage(ADSLOG_MSGTYPE_ERROR, 'OOSC3', 'PropertyBuffer: Uninitialized property type!');
		
	ELSIF (ValidateInst()) THEN
		// Initialize COV-Trigger:
		IF (fbRefObject^.SyncPropertyCOV(ePropertyID, ADR(bChangeTrig))) THEN
			// Initialize property:
			IF (nUsedSize = 0) THEN
				// Initial value has defenitly to be read from stack:
				bReady := SUCCEEDED(ReadValue());
			ELSE
				CASE (eSyncMode) OF
					eSync_ToSupplement,
					eFullSync_InitPLC:
						bReady := SUCCEEDED(WriteValue());
				ELSE
					bReady := SUCCEEDED(ReadValue());
				END_CASE
			END_IF
		END_IF
	END_IF
END_IF
END_METHOD

METHOD ResetValue
nUsedSize := 0;

ValidateInst();
END_METHOD

END_FUNCTION_BLOCK

// POUs/Local/Objects/[Internal]/Property/Buffer/Base/FB_BACnet_BaseArrayBuffer
FUNCTION_BLOCK INTERNAL FB_BACnet_BaseArrayBuffer EXTENDS FB_BACnet_BasePropertyBuffer
VAR CONSTANT
	{attribute 'hide'}
	nBACnet_EntryCount	: UINT	:= 256;
	
	// Hint:
	// > [BufferSize] := (nBACnet_EntryCount * [EntrySize])
END_VAR

SUPER^();

END_FUNCTION_BLOCK

// POUs/Local/Objects/[Internal]/Property/Buffer/Base/FB_BACnet_BasePropertyLogBuffer
FUNCTION_BLOCK FB_BACnet_BasePropertyLogBuffer EXTENDS FB_BACnet_BasePropertyBuffer

SUPER^();

METHOD OnObjectStateChanged
VAR_INPUT
	tState : TCOM_STATE;
END_VAR
VAR
	eSyncMode : E_BA_FullSyncMode := eFullSync_InitPLC;
END_VAR
IF (tState = tSyncState) THEN
	IF (ePropertyID = E_BACnetPropIdentifier.PropInvalid) THEN
		F_BA_LogMessage(ADSLOG_MSGTYPE_ERROR, 'OOSC8', 'PropertyBuffer: Uninitialized property type!');
		
	ELSIF (ValidateInst()) THEN
		// Initialize COV-Trigger:
		IF (fbRefObject^.SyncPropertyCOV(ePropertyID, ADR(bChangeTrig))) THEN
			// Initialize property:
			IF (nUsedSize = 0) THEN
				IF fbRefObject^.bIsReused THEN
					// Reset stack value:
					bReady := SUCCEEDED(fbRefObject^.WritePropertyUDInt(E_BACnetPropIdentifier.PropTotalRecordCount,0));
				ELSE
					// Initial value has defenitly to be read from stack:
					bReady := SUCCEEDED(ReadValue());
				END_IF
			ELSE
				IF fbRefObject^.bIsReused THEN
					bReady := SUCCEEDED(ReadValue());
				ELSE
					bReady := SUCCEEDED(WriteValue());
				END_IF
			END_IF
		END_IF
	END_IF
END_IF
END_METHOD

END_FUNCTION_BLOCK

// POUs/Local/Objects/[Internal]/Property/Buffer/FB_BACnet_DateListBuffer
FUNCTION_BLOCK INTERNAL FB_BACnet_DateListBuffer EXTENDS FB_BACnet_BaseListBuffer

SUPER^();

METHOD FB_init : BOOL
VAR_INPUT
	bInitRetains : BOOL; // if TRUE, the retain variables are initialized (warm start / cold start)
	bInCopyCode : BOOL;  // if TRUE, the instance afterwards gets moved into the copy code (online change)
END_VAR
ePropertyID := E_BACnetPropIdentifier.PropDateList;
END_METHOD

END_FUNCTION_BLOCK

// POUs/Local/Objects/[Internal]/Property/Buffer/FB_BACnet_EventLogBuffer
FUNCTION_BLOCK INTERNAL FB_BACnet_EventLogBuffer EXTENDS FB_BACnet_BasePropertyBuffer
VAR PERSISTENT
	aBuffer : ARRAY[1 .. nBACnet_BufferSize] OF BYTE;
END_VAR
VAR CONSTANT
	{attribute 'hide'}
	{attribute 'parameterUnit':= 'byte'}
	nBACnet_EntrySize	: UDINT	:= 376;
	{attribute 'hide'}
	nBACnet_EntryCount	: UDINT	:= BACnet_Param.nLog_BufferEntryCount;
	
	{attribute 'hide'}
	nBACnet_BufferSize	: UDINT	:= (nBACnet_EntrySize * nBACnet_EntryCount);
END_VAR

SUPER^();

METHOD PROTECTED ValidateInst : BOOL
nBufferSize := SIZEOF(aBuffer);
pBufferValue := ADR(aBuffer);

ValidateInst := SUPER^.ValidateInst();
END_METHOD

METHOD FB_init : BOOL
VAR_INPUT
	bInitRetains : BOOL; // if TRUE, the retain variables are initialized (warm start / cold start)
	bInCopyCode : BOOL;  // if TRUE, the instance afterwards gets moved into the copy code (online change)
END_VAR
ePropertyID := E_BACnetPropIdentifier.PropLogBuffer;
END_METHOD

END_FUNCTION_BLOCK

// POUs/Local/Objects/[Internal]/Property/Buffer/FB_BACnet_ExceptionScheduleBuffer
FUNCTION_BLOCK INTERNAL FB_BACnet_ExceptionScheduleBuffer EXTENDS FB_BACnet_BaseListBuffer

SUPER^();

METHOD FB_init : BOOL
VAR_INPUT
	bInitRetains : BOOL; // if TRUE, the retain variables are initialized (warm start / cold start)
	bInCopyCode : BOOL;  // if TRUE, the instance afterwards gets moved into the copy code (online change)
END_VAR
ePropertyID := E_BACnetPropIdentifier.PropExceptionSchedule;
END_METHOD

END_FUNCTION_BLOCK

// POUs/Local/Objects/[Internal]/Property/Buffer/FB_BACnet_TLMBuffer
FUNCTION_BLOCK INTERNAL FB_BACnet_TLMBuffer EXTENDS FB_BACnet_BasePropertyLogBuffer
VAR PERSISTENT
	aBuffer : ARRAY[1 .. nBACnet_BufferSize] OF BYTE;
END_VAR
VAR CONSTANT
	{attribute 'hide'}
	{attribute 'parameterUnit':= 'byte'}
	nBACnet_HeaderSize		: UINT	:= 20;
	{attribute 'hide'}
	{attribute 'parameterUnit':= 'byte'}
	nBACnet_EntrySize		: UINT	:= 5;
	{attribute 'hide'}
	nBACnet_EntryCount		: UINT	:= TO_UINT(BACnet_Param.nLog_BufferEntryCount);
	{attribute 'hide'}
	nBACnet_EntryItemCount	: UINT	:= 100;
	
	{attribute 'hide'}
	nBACnet_BufferSize		: UINT	:= nBACnet_HeaderSize + ((nBACnet_EntrySize * nBACnet_EntryCount) * nBACnet_EntryItemCount);
END_VAR

SUPER^();

METHOD PROTECTED ValidateInst : BOOL
nBufferSize := SIZEOF(aBuffer);
pBufferValue := ADR(aBuffer);

ValidateInst := SUPER^.ValidateInst();
END_METHOD

METHOD ResetValue
VAR
	stTimestamp : POINTER TO ST_BA_DateTime;
END_VAR
SUPER^.ResetValue();

// Write one log-entry "log-disabled" to buffer:
MemSetULINT(16#0000000100000020, nUsedSize);
MemSetUDINT(16#00000003, nUsedSize);

(*
stTimestamp := (pBufferValue+nUsedSize);
stTimestamp^ := F_GetCurrentTime();
nUsedSize := (nUsedSize+SIZEOF(ST_DateTime));
*)
MemSetULINT(16#51152607021D0177, nUsedSize);

MemSetUDINT(16#00000000, nUsedSize);
MemSetULINT(16#0000000000000008, nUsedSize);
MemSetULINT(16#0000800500000000, nUsedSize);
END_METHOD

METHOD FB_init : BOOL
VAR_INPUT
	bInitRetains : BOOL; // if TRUE, the retain variables are initialized (warm start / cold start)
	bInCopyCode : BOOL;  // if TRUE, the instance afterwards gets moved into the copy code (online change)
END_VAR
ePropertyID := E_BACnetPropIdentifier.PropLogBuffer;
END_METHOD

END_FUNCTION_BLOCK

// POUs/Local/Objects/[Internal]/Property/Buffer/FB_BACnet_TrendLogBuffer
FUNCTION_BLOCK INTERNAL FB_BACnet_TrendLogBuffer EXTENDS FB_BACnet_BasePropertyLogBuffer
VAR PERSISTENT
	aBuffer : ARRAY[1 .. nBACnet_BufferSize] OF BYTE;
END_VAR
VAR CONSTANT
	{attribute 'parameterUnit':= 'byte'}
	nBACnet_EntrySize	: UDINT	:= 56;
	nBACnet_EntryCount	: UDINT	:= BACnet_Param.nLog_BufferEntryCount;
	nBACnet_BufferSize	: UDINT	:= (nBACnet_EntrySize * nBACnet_EntryCount);
END_VAR

SUPER^();

METHOD PROTECTED ValidateInst : BOOL
nBufferSize := SIZEOF(aBuffer);
pBufferValue := ADR(aBuffer);

ValidateInst := SUPER^.ValidateInst();
END_METHOD

METHOD ResetValue
VAR
	stTimestamp : POINTER TO ST_BA_DateTime;
END_VAR
SUPER^.ResetValue();

// Write one log-entry "log-disabled" to buffer:
MemSetULINT(16#0000000100000020, nUsedSize);
MemSetUDINT(16#00000003, nUsedSize);

(*
stTimestamp := (pBufferValue+nUsedSize);
stTimestamp^ := F_GetCurrentTime();
nUsedSize := (nUsedSize+SIZEOF(ST_DateTime));
*)
MemSetULINT(16#51152607021D0177, nUsedSize);

MemSetUDINT(16#00000000, nUsedSize);
MemSetULINT(16#0000000000000008, nUsedSize);
MemSetULINT(16#0000800500000000, nUsedSize);
END_METHOD

METHOD FB_init : BOOL
VAR_INPUT
	bInitRetains : BOOL; // if TRUE, the retain variables are initialized (warm start / cold start)
	bInCopyCode : BOOL;  // if TRUE, the instance afterwards gets moved into the copy code (online change)
END_VAR
ePropertyID := E_BACnetPropIdentifier.PropLogBuffer;
END_METHOD

END_FUNCTION_BLOCK

// POUs/Local/Objects/Experimental/FB_BACnet_ExpEventLog
{attribute 'hide'}	// (BETA) ...FB is only for testing!



FUNCTION_BLOCK FB_BACnet_ExpEventLog EXTENDS FB_BACnet_BaseTLog

VAR_INPUT CONSTANT PERSISTENT
	{region 'Fixed Parameters'}
		// (BETA) ... Implement "EventLogBuffer"-Property
		//{attribute 'hide'}
		//{attribute 'parameterCategory':='Value'}
		//aLogBuffer : ARRAY [1 .. BACnet_Param.nEventLog_BufferEntryCount] OF ST_BACnet_EventLogEntry;
	{endregion}
END_VAR

END_FUNCTION_BLOCK

// POUs/Local/Objects/Experimental/FB_BACnet_ExpTLM
{attribute 'hide'}	// (BETA) ...FB is only for testing!


FUNCTION_BLOCK FB_BACnet_ExpTLM EXTENDS FB_BACnet_BaseTLog
VAR_INPUT CONSTANT PERSISTENT
	{region 'Fixed Parameters'}
		// (BETA) ... Implement "LogBuffer(Multiple)"-Property
		//{attribute 'hide'}
		//{attribute 'parameterCategory':='Value'}
		//aLogBuffer : ARRAY [1 .. BACnet_Param.nTLM_ArraySize] OF ST_BACnet_TLMEntry;
	{endregion}
END_VAR
VAR PERSISTENT
	{region 'SubInit'}
		// (BETA) ... Implement "DeviceObjPropRef(Multiple)"-Property
		// ...
	{endregion}
END_VAR
VAR
	{region 'Buffers'}
		{attribute 'conditionalshow'}
		fbLogBuffer					: FB_BACnet_TLMBuffer			:= (iRefObject := THIS^);
	{endregion}
END_VAR

// Synchronize Buffers:
fbLogBuffer();

SUPER^();

METHOD PROTECTED OnObjectStateChanged
SUPER^.OnObjectStateChanged();

// Synchronize:
fbLogBuffer.OnObjectStateChanged(tState);

CASE (tState) OF
	TCOM_STATE.TCOM_STATE_PREOP:
		;
	
	TCOM_STATE.TCOM_STATE_SAFEOP:
		;

	TCOM_STATE.TCOM_STATE_OP:
		;
		
END_CASE
END_METHOD

METHOD FB_init : BOOL
VAR_INPUT
	bInitRetains : BOOL; // if TRUE, the retain variables are initialized (warm start / cold start)
	bInCopyCode : BOOL;  // if TRUE, the instance afterwards gets moved into the copy code (online change)
END_VAR
eObjectType := E_BACnetObjType.ObjTrendLogMultiple;
END_METHOD

END_FUNCTION_BLOCK

// POUs/Local/Objects/Experimental/FB_BACnet_ExpTLog
{attribute 'hide'}	// (BETA) ...FB is only for testing!


FUNCTION_BLOCK FB_BACnet_ExpTLog EXTENDS FB_BACnet_BaseTLog
VAR_INPUT CONSTANT PERSISTENT
	{region 'Variable Parameters'}
		{attribute 'parameterCategory':='Value'}
		aLogBuffer : T_BACnet_TLogBuffer;
		{attribute 'parameterCategory':='Value'}
		bWriteLogBuffer : BOOL;
			 
		{attribute 'parameterCategory':='Config'}
		stObjectPropertyReference : ST_BACnet_ObjectPropertyReference;
	{endregion}
END_VAR
VAR
	{region 'COV'}
		bLogBufferChanged			: BOOL;
	{endregion}
END_VAR

IF (bWriteLogBuffer) THEN
	{warning disable C0196}
	WritePropertyLogBuffer(aLogBuffer);
	{warning restore C0196}
	
	bWriteLogBuffer := FALSE;
END_IF
IF (bLogBufferChanged) THEN
	{warning disable C0196}
	ReadPropertyLogBuffer(aLogBuffer);
	{warning restore C0196}
	
	bLogBufferChanged := FALSE;
END_IF

SUPER^();

//check PLC Buffer for last valid record entry
METHOD PRIVATE Trend_LastPlcTrendEntry : BOOL
VAR_INPUT
	_pTrendEntry					: POINTER TO ST_BA_TrendEntry;
END_VAR
Trend_LastPlcTrendEntry := 	(_pTrendEntry^.dtTime.stDate.eMonth = E_BA_MONTH.Invalid) AND 
							(_pTrendEntry^.dtTime.stDate.eDayOfWeek = E_BA_WEEKDAY.Invalid) AND
							(_pTrendEntry^.eType = E_BA_TRENDENTRYTYPE.Invalid);
END_METHOD

//Trend_NextLogRecord Springe zum nächsten LogEintrag und verschiebe Pointer um länge des Logrecords
METHOD PRIVATE Trend_NextLogDatum : BOOL
VAR_IN_OUT
	_pLbDatumList					: POINTER TO ST_BACnet_LogDatumList;
	_cbTotalBuf						: UDINT;
END_VAR
VAR
	_cbTmpSize						: UDINT;
END_VAR
Trend_NextLogDatum := ((_pLbDatumList^.nEntrySize AND 16#80000000) = 16#80000000);

_cbTmpSize := F_BACnet_AlignedSize(_pLbDatumList^.nEntrySize AND 16#7FFFFFFF) + SIZEOF(_pLbDatumList^.nEntrySize) + SIZEOF(_pLbDatumList^.reserved);
_pLbDatumList	:= _pLbDatumList + _cbTmpSize;
_cbTotalBuf := _cbTotalBuf + _cbTmpSize;
END_METHOD

//Trend_NextLogRecord Springe zum nächsten LogEintrag und verschiebe Pointer um länge des Logrecords
METHOD PRIVATE Trend_NextLogRecord : BOOL
VAR_IN_OUT
	_pLbRecordList					: POINTER TO ST_BACnet_LogRecordList;
	_cbTotalBuf						: UDINT;
END_VAR
VAR_INPUT
	bIndicateLastEntry				: BOOL		:= FALSE;
END_VAR
VAR
	_cbTmpSize						: UDINT;
END_VAR
Trend_NextLogRecord := ((_pLbRecordList^.nEntrySize AND 16#80000000) = 16#80000000);

_cbTmpSize := F_BACnet_AlignedSize(_pLbRecordList^.nEntrySize AND 16#7FFFFFFF) + SIZEOF(_pLbRecordList^.nEntrySize) + SIZEOF(_pLbRecordList^.nSequence);
IF (bIndicateLastEntry) THEN
	_pLbRecordList^.nEntrySize := (_pLbRecordList^.nEntrySize AND 16#7FFFFFFF); // Set Bit 31 to false to signal this is last Record
ELSE
	_pLbRecordList	:= _pLbRecordList + _cbTmpSize;	// move pointer
END_IF
_cbTotalBuf := _cbTotalBuf + _cbTmpSize;	// calculate total buffersize
END_METHOD

METHOD PROTECTED OnObjectStateChanged
SUPER^.OnObjectStateChanged();

CASE (tState) OF
	TCOM_STATE.TCOM_STATE_PREOP:
		// SyncHandler:
		RequestSyncHandlers(1, 0);
	
	TCOM_STATE.TCOM_STATE_SAFEOP:
		;

	TCOM_STATE.TCOM_STATE_OP:
		// Validate referred property:
		IF (ValidateReference(stObjectPropertyReference.iObject, stObjectPropertyReference.tObjectID, 16#FF)) THEN
			ObjectPropertyReference := stObjectPropertyReference;
		END_IF
		
		SyncPropertyCOV(E_BACnetPropIdentifier.PropLogBuffer, ADR(bLogBufferChanged));
		
END_CASE
END_METHOD

METHOD ReadPropertyLogBuffer : HRESULT
VAR_IN_OUT
	aLogBuffer						: ARRAY [*] OF ST_BA_TrendEntry;
END_VAR
VAR
	// general
	_nLength						: DINT;
	_cbTotalBuf						: UDINT;
	_cbDatumBuf						: UDINT;
	// Pointer_to_...
	_pLbRecordList					: POINTER TO ST_BACnet_LogRecordList;								// Pointer Log buffer - LogRecordList of LogBuffer
	_pLbLogRec						: POINTER TO ST_BACnet_LogRecord;									// Pointer Log Buffer - LogRecord of LogRecordList
	_pLbDatumList					: POINTER TO ST_BACnet_LogDatumList;								// Pointer Log Buffer - DatumList of LogRecord
	// indexvariables
	_nRecCount						: UDINT;															// Log record entry - Record list
	_nRecDatumCount					: UDINT;															// Log record entry - datum list
	_nMaxSeq						: DWORD;
	// sizeinfos		
	_nPOffsetEntrySize				: DWORD;	//Offset für verschiebung des Pointers (Log Entrysize + Header)
	_nPOffsetRecordSize				: DWORD;	//Offset für verschiebung des Pointers (Log Entrysize + Header)
END_VAR
IF (ipObj = 0) THEN
	_hResult := E_FAIL;
ELSE
	_nLength := SIZEOF(BACnet_Globals.aDefaultBuffer);
	_hResult := ReadProperty(E_BACnetPropIdentifier.PropLogBuffer, ADR(BACnet_Globals.aDefaultBuffer), ADR(_nLength));
	
	IF (SUCCEEDED(_hResult)) THEN
		IF (_nLength > 0) THEN
			MEMSET(aLogBuffer, 0, TO_UDINT(F_BA_TrendBufferSize(aLogBuffer)));	// clear current PLC LogBuffer	
			// Point to first data:
			_pLbRecordList := ADR(BACnet_Globals.aDefaultBuffer);
			_cbTotalBuf := 0;
			_nRecCount := 0;
			_nRecDatumCount := 0;
			_nMaxSeq := 0;
			
			// Show Buffercontent
//(* DEBUG *)	F_BA_Print('[ST_BACnet_LogRecordList] frist Readout', _pLbRecordList, TO_UINT(_nLength), TRUE, 40);	
			_pLbLogRec := ADR(_pLbRecordList^.listEntry); // Pointer to first Entry  of LogRecord of logrecordlist
			
			// ----------------------------------------------------------------------------------------------------------
			// Parsing Logbuffer
			IF (_pLbLogRec <> 0) THEN
				// iterate  parsing of logbuffer until length of Entrysize = 0 (no more entrys )
				// identify LogRecords from logrecordlist
				REPEAT
					// Determine the length of the pointer offset: Value of Entrysize + header length (2 Dwords)
					_nPOffsetEntrySize := (_pLbRecordList^.nEntrySize AND 16#7FFFFFFF);
					
					IF (_nPOffsetEntrySize > 0) THEN
						_pLbLogRec 		:= ADR(_pLbRecordList^.listEntry);	// Pointer to first Entry  of LogRecord of logrecordlist
						_pLbDatumList	:= ADR(_pLbLogRec^.logDatum);		// Pointer to first Entry of Datumlist of LogRecord
						// Next Logentry and Sequence
						_nRecCount := _nRecCount+1;
						_nMaxSeq := _pLbRecordList^.nSequence;

//(* DEBUG *)			F_BA_LogMessage3(ADSLOG_MSGTYPE_LOG, 'RPLB45', '%s (Nr.: %d, SeqNr.: %d in TotalRecordCount)',F_STRINGEx('LogRecord: '), F_UDINT(_nRecCount), F_DWORD(_nMaxSeq));
//(* DEBUG *)			F_BA_Print('[ST_BACnet_LogRecord] ',_pLbLogRec, TO_UINT(_nPOffsetEntrySize), TRUE, TO_UINT(_nPOffsetEntrySize));						
						
						// [BACStac Logbuffer -> PLC Logbuffer] Sync/Fill PLC Logbuffer
						// Insert Current Logrecord from ST_BACnet_LogRecordList into aLogBuffer
						IF ( (_pLbDatumList <> 0) AND (_nRecCount > 0) ) THEN
							// Insert Timestamp
							aLogBuffer[_nRecCount].dtTime := _pLbLogRec^.timestamp;
							// Insert Statusflags
							aLogBuffer[_nRecCount].stState := F_BACnet_StatusFlags(TO_WORD(_pLbLogRec^.statusFlags));
								//aLogBuffer[_nRecCount].stState.bInAlarm		:= TO_BOOL(_pLbLogRec^.statusFlags AND 16#8000);
								//aLogBuffer[_nRecCount].stState.bFault			:= TO_BOOL(_pLbLogRec^.statusFlags AND 16#4000);
								//aLogBuffer[_nRecCount].stState.bOverridden	:= TO_BOOL(_pLbLogRec^.statusFlags AND 16#2000);
								//aLogBuffer[_nRecCount].stState.bOutOfService	:= TO_BOOL(_pLbLogRec^.statusFlags AND 16#1000);
							// Logdatum (Value)
							MEMCPY(ADR(aLogBuffer[_nRecCount].uValue), ADR(_pLbDatumList^.listEntry.aData[0]), SIZEOF(_pLbDatumList^.listEntry.aData[0]));									
							// Typecasting (Logdatum Type / Choice)
							CASE (_pLbLogRec^.logDatum.listEntry.choice) OF 
								E_BACnet_LogRecordChoice.eLogStatus:	(*	[0] BACnetLogStatus *)	
									aLogBuffer[_nRecCount].eType := E_BA_TrendEntryType.eEvent;													
									CASE _pLbDatumList^.listEntry.aData[0] OF 
										16#0005: aLogBuffer[_nRecCount].uValue.eEvent := E_BA_TrendEntryEvent.eStart;
										16#2005: aLogBuffer[_nRecCount].uValue.eEvent := E_BA_TrendEntryEvent.eInterrupted;
										16#4005: aLogBuffer[_nRecCount].uValue.eEvent := E_BA_TrendEntryEvent.eBufferPurged;
										16#8005: aLogBuffer[_nRecCount].uValue.eEvent := E_BA_TrendEntryEvent.eStop; // Stop/Disabled
									ELSE
										;// value from MEMCPY operation before 
									END_CASE								
								E_BACnet_LogRecordChoice.eBooleanValue: (*  [1] BOOL, *)
									aLogBuffer[_nRecCount].eType := E_BA_TrendEntryType.eBinary;
								E_BACnet_LogRecordChoice.eRealValue:	(*  [2] REAL *)
									aLogBuffer[_nRecCount].eType := E_BA_TrendEntryType.eAnalog;	
								E_BACnet_LogRecordChoice.eEnumValue:	(*	[3] ENUMERATED, __ Optionally limited to 32 bits *)
									aLogBuffer[_nRecCount].eType := E_BA_TrendEntryType.eMultistate;								
								E_BACnet_LogRecordChoice.eUnsignedValue:(*	[4] Unsigned, __ Optionally limited to 32 bits *)
									aLogBuffer[_nRecCount].eType := E_BA_TrendEntryType.eMultistate;								
							ELSE
								aLogBuffer[_nRecCount].eType := E_BA_TrendEntryType.Invalid;
							END_CASE				
													
						END_IF					
						// ----------------------------------------------------------------------------------------------------------
//possibly unnecessary	// calculate number of Elements of Logdatum  from Logdatumlist
						IF (_pLbDatumList <> 0) THEN
							_nPOffsetRecordSize := (_pLbDatumList^.nEntrySize AND 16#7FFFFFFF);
							_nRecDatumCount := 0;
							REPEAT 
								_nRecDatumCount := _nRecDatumCount+1;
								IF (NOT	Trend_NextLogDatum(_pLbDatumList, _cbDatumBuf)) THEN
									EXIT;
								END_IF
							UNTIL	(_nRecDatumCount > 4)// Buffer full
							END_REPEAT
						END_IF
						
					END_IF
					
					// Next LogRecordEntry ?
					// Trend_NextLogRecord update Pointer to next logrecord by size of Logrecord
					IF (NOT	Trend_NextLogRecord(_pLbRecordList, _cbTotalBuf, FALSE)) THEN
						EXIT;	//leave
					END_IF
															
				UNTIL (		(_nRecCount >= (BACnet_Globals.nDataField_MaxLogBufferEntries + 1)) (* result buffer full *)
						OR	(_pLbRecordList >= (ADR(BACnet_Globals.aDefaultBuffer) + _nLength)) (* ads buffer ending reached *)
					)
				END_REPEAT
			END_IF
			
//(* DEBUG *)	F_BA_LogMessage3(ADSLOG_MSGTYPE_LOG, 'RPLB_100', '%s ( %d of %d in TotalRecordCount)',F_STRINGEx('Valid Log Records: '), F_UDINT(_nRecCount) ,F_UDINT(_nMaxSeq) );			
					
		END_IF
	ELSE
		iOwner.LogMsg.Show1(ADSLOG_MSGTYPE_ERROR, 'RLB_400', 'Failed to read log buffer property! (Error 0x%x)', F_DINT(_hResult), TRUE);
	END_IF
END_IF


ReadPropertyLogBuffer := _hResult;
END_METHOD

METHOD WritePropertyLogBuffer : HRESULT
VAR_IN_OUT
	aLogBuffer						: ARRAY [*] OF ST_BA_TrendEntry;
END_VAR
VAR
	// general
	_nLength						: DINT;
	_cbTotalBuf						: UDINT;

	// Pointer_to_...
	_pLbRecordList					: POINTER TO ST_BACnet_LogRecordList;								// Pointer Log buffer - LogRecordList of LogBuffer
	_pLbLogRec						: POINTER TO ST_BACnet_LogRecord;									// Pointer Log Buffer - LogRecord of LogRecordList
	_pLbDatumList					: POINTER TO ST_BACnet_LogDatumList;								// Pointer Log Buffer - DatumList of LogRecord
	// indexvariables
	_nRecCount						: UDINT;															// Log record entry - Record list
	
	_nMaxSeq						: DWORD;
	// sizeinfos	
	_nPOffsetEntrySize				: DWORD;	//Offset für verschiebung des Pointers (Log Entrysize + Header)
END_VAR
IF (ipObj = 0) THEN
	_hResult := E_FAIL;
ELSE
	_hResult := S_OK;

	// Point to first data:
	_nLength := SIZEOF(BACnet_Globals.aDefaultBuffer);
	_pLbRecordList := ADR(BACnet_Globals.aDefaultBuffer);
	_cbTotalBuf := 0;
	
	IF (SUCCEEDED(_hResult)) THEN
			
		_nRecCount := 1;
		_nPOffsetEntrySize := 16#80000020; // Set Fag (nextlogrecord) [b31], Set Entrysize (length) of Logrecord [32 Byte] 
		_pLbRecordList^.nEntrySize := _nPOffsetEntrySize;
		
		_nMaxSeq := BACnet_Globals.nDataField_MaxLogBufferEntries+1;
		
		// ----------------------------------------------------------------------------------------------------------
		// Parsing PLC Logbuffer
		REPEAT 
			// set pointer
			_pLbRecordList^.nEntrySize := _nPOffsetEntrySize;		//Calculate size for next log entry, set bit 31 because further elements will follow			
			_pLbLogRec 		:= ADR(_pLbRecordList^.listEntry);	//Pointer to first Entry  of LogRecord of logrecordlist
			_pLbDatumList	:= ADR(_pLbLogRec^.logDatum);		//Pointer to first Entry of Datumlist of LogRecord
			// set sequencenumber of logentry
			_pLbRecordList^.nSequence := _nRecCount;
			
			// [PLC Logbuffer -> BACStac Logbuffer ] 
			// Constructing Sync/Fill Stac Logbuffer
			IF ( (_pLbDatumList <> 0) AND (_nRecCount > 0) ) THEN
				// Timestamp
				_pLbLogRec^.timestamp := aLogBuffer[_nRecCount].dtTime;
				// Insert Statusflags
				_pLbLogRec^.statusFlags := F_BACnet_GetStatusFlagsData(aLogBuffer[_nRecCount].stState);
				// Logdatum (Header)
				_pLbDatumList^.nEntrySize := 16#08;//SIZEOF(_pLbDatumList^.listEntry.aData[0]); //Header Logdatum List set length
				// Logdatum (Value) 
				MEMCPY(ADR(_pLbDatumList^.listEntry.aData[0]), ADR(aLogBuffer[_nRecCount].uValue), SIZEOF(_pLbDatumList^.listEntry.aData[0]));									
				// Typecasting (Logdatum Type / Choice / Valid Fields)
				CASE (aLogBuffer[_nRecCount].eType) OF
					E_BA_TrendEntryType.eEvent: 
						_pLbLogRec^.validFields := 16#03; 	//Valid Fields Timestamp and Logrecord
						_pLbLogRec^.statusFlags := 16#00;	//Reset Statusflags	
						_pLbLogRec^.logDatum.listEntry.choice := E_BACnet_LogRecordChoice.eLogStatus;	(* BACnetLogStatus *)
						// Flags setzen finde ich besser aber die daten liegen nunmal nicht mehr vor
						CASE (aLogBuffer[_nRecCount].uValue.eEvent) OF 
							E_BA_TrendEntryEvent.eStart: 		_pLbDatumList^.listEntry.aData[0] := 16#0005;
							E_BA_TrendEntryEvent.eInterrupted: 	_pLbDatumList^.listEntry.aData[0] := 16#2005;
							E_BA_TrendEntryEvent.eBufferPurged:	_pLbDatumList^.listEntry.aData[0] := 16#4005;
							E_BA_TrendEntryEvent.eStop: 		_pLbDatumList^.listEntry.aData[0] := 16#8005;
						END_CASE
					E_BA_TrendEntryType.eBinary:
						_pLbLogRec^.validFields := 16#07;
						_pLbLogRec^.logDatum.listEntry.choice := E_BACnet_LogRecordChoice.eBooleanValue; (*  BOOL, *)
					E_BA_TrendEntryType.eAnalog:
						_pLbLogRec^.validFields := 16#07;	
						_pLbLogRec^.logDatum.listEntry.choice := E_BACnet_LogRecordChoice.eRealValue;	(*  REAL, *)
					E_BA_TrendEntryType.eMultistate:
						_pLbLogRec^.validFields := 16#07;								
						_pLbLogRec^.logDatum.listEntry.choice := E_BACnet_LogRecordChoice.eUnsignedValue;	(*  ENUMERATED, __ Optionally limited TO 32 bits *)	
				ELSE
					_pLbLogRec^.logDatum.listEntry.choice := E_BACnet_LogRecordChoice.eLogStatus;
				END_CASE
			END_IF
					
//(* DEBUG *)	F_BA_LogMessage3(ADSLOG_MSGTYPE_LOG, 'WPLB_10', '%s (Nr.: %d, SeqNr.: %d in TotalRecordCount)',F_STRINGEx('LogRecord: '), F_UDINT(_nRecCount), F_DWORD(_pLbRecordList^.nSequence));
//(* DEBUG *)	F_BA_Print('[ST_BACnet_LogRecord] ',_pLbLogRec, TO_UINT(_nPOffsetEntrySize), TRUE, TO_UINT(_nPOffsetEntrySize));
			
			// Next LogRecordEntry		
			_nRecCount := _nRecCount + 1;
			// Check whether the last entry in the PLC buffer has been reached
			IF (Trend_LastPlcTrendEntry(ADR(aLogBuffer[_nRecCount]))) THEN				
				// Last LogRecordEntry
				Trend_NextLogRecord(_pLbRecordList, _cbTotalBuf, TRUE ); //Signal Trend Last Record set flag (b31) for last listentry on the current header of logentry			
				EXIT;	// leave
			ELSE
				// Trend_NextLogRecord update Pointer to next logrecord by size of Logrecord
				Trend_NextLogRecord(_pLbRecordList, _cbTotalBuf, FALSE );
			END_IF
			
		UNTIL	(_nRecCount >= (BACnet_Globals.nDataField_MaxLogBufferEntries + 1) )// Buffer full
		END_REPEAT
		
//(* DEBUG *)	F_BA_LogMessage3(ADSLOG_MSGTYPE_LOG, 'WPLB_20', '%s ( %d of %d in TotalRecordCount)',F_STRINGEx('Valid Log Records: '), F_UDINT(_pLbRecordList^.nSequence) ,F_UDINT(_nMaxSeq) );			 
//(* DEBUG *)	_pLbRecordList := ADR(BACnet_Globals.aDefaultBuffer);//Pointer to  Start (Logentry 1) check current Buffer output 
//(* DEBUG *)	F_BA_Print('[ST_BACnet_LogRecordList]  Write Buffer', _pLbRecordList, TO_UINT(_cbTotalBuf), TRUE, 40);	

	END_IF
	
	// Write data:
	_hResult := WriteProperty(E_BACnetPropIdentifier.PropLogBuffer, ADR(BACnet_Globals.aDefaultBuffer), TO_DINT(_cbTotalBuf));
	
END_IF	

WritePropertyLogBuffer := _hResult;
END_METHOD

PROPERTY ObjectPropertyReference : ST_BACnet_ObjectPropertyReference
GET
ObjectPropertyReference := stObjectPropertyReference;
END_GET
SET
stObjectPropertyReference := ObjectPropertyReference;

WritePropertyReference(E_BACnetPropIdentifier.PropLogDeviceObjectProperty, stObjectPropertyReference);
END_SET
END_PROPERTY

METHOD FB_init : BOOL
VAR_INPUT
	bInitRetains : BOOL; // if TRUE, the retain variables are initialized (warm start / cold start)
	bInCopyCode : BOOL;  // if TRUE, the instance afterwards gets moved into the copy code (online change)
END_VAR
eObjectType := E_BACnetObjType.ObjTrendLog;
END_METHOD

END_FUNCTION_BLOCK

